	PUMP_STATUS:	(* Status and Fault *)
		Modbus.MB_Lock := TRUE;
		Modbus.MB_Query.SlaveAddress := Address;
		Modbus.MB_Query.FunctionCode := 3;
		ModBus.MB_Query.Read_StartAddress := 201;
		ModBus.MB_Query.Read_Quantity := 2;
		ModBus.MB_Start := TRUE;

		state := PUMP_DATA;

	PUMP_DATA:	(* Pump data *)
		IF NOT ModBus.MB_Start THEN
			IF ModBus.MB_MASTER.bInterfaceError<>0 OR ModBus.MB_MASTER.MB_Error<>0 THEN
				state := ERROR_STATE;
			ELSE
				DataPump.PumpStatus := ModBus.MB_Resp.Data[0];
				DataPump.PumpFault	:= WORD_TO_BOOL(ModBus.MB_Resp.Data[1]);

				ModBus.MB_Query.Read_StartAddress := 210;
				ModBus.MB_Query.Read_Quantity := 12;
				ModBus.MB_Start := TRUE;

				state := PUMP_ALARMS;
			END_IF
		END_IF

	PUMP_ALARMS: (* Historical alarms *)
		IF NOT ModBus.MB_Start THEN
			IF ModBus.MB_MASTER.bInterfaceError<>0 OR ModBus.MB_MASTER.MB_Error<>0 THEN
				state := ERROR_STATE;
			ELSE
				DataPump.PumpBoardTemp 	:= WORD_TO_INT(ModBus.MB_Resp.Data[0]);
				DataPump.PumpVoltage	:= ModBus.MB_Resp.Data[2];
				DataPump.PumpCurrent	:= ModBus.MB_Resp.Data[3];
				DataPump.PumpRPM		:= ModBus.MB_Resp.Data[5];
				DataPump.PumpPower		:= ModBus.MB_Resp.Data[6];
				DataPump.PumpOpTime		:= BUILD_16TO32(ADR(ModBus.MB_Resp.Data[7]));
				DataPump.PumpHead		:= ModBus.MB_Resp.Data[9];
				DataPump.PumpFlow		:= ModBus.MB_Resp.Data[10];
				DataPump.PumpLiqTemp	:= WORD_TO_INT(ModBus.MB_Resp.Data[11]);


				ModBus.MB_Query.Read_StartAddress := 230;
				ModBus.MB_Query.Read_Quantity := 15;
				ModBus.MB_Start := TRUE;

				state := PUMP_END_READ;
			END_IF
		END_IF

	PUMP_END_READ:	(* Read alarms *)
		IF NOT ModBus.MB_Start THEN
			IF ModBus.MB_MASTER.bInterfaceError<>0 OR ModBus.MB_MASTER.MB_Error<>0 THEN
				state := ERROR_STATE;
			ELSE
				DataPump.PumpAlarm[0] := ModBus.MB_Resp.Data[0];
				DataPump.PumpAlarm[1] := ModBus.MB_Resp.Data[1];
				DataPump.PumpAlarm[2] := ModBus.MB_Resp.Data[2];
				DataPump.PumpAlarm[3] := ModBus.MB_Resp.Data[3];
				DataPump.PumpAlarm[4] := ModBus.MB_Resp.Data[4];
				DataPump.PumpAlarm[5] := ModBus.MB_Resp.Data[5];
				DataPump.PumpAlarm[6] := ModBus.MB_Resp.Data[6];
				DataPump.PumpAlarm[7] := ModBus.MB_Resp.Data[7];
				DataPump.PumpAlarm[8] := ModBus.MB_Resp.Data[8];
				DataPump.PumpAlarm[9] := ModBus.MB_Resp.Data[9];
				DataPump.PumpAlarm[10] := ModBus.MB_Resp.Data[10];
				DataPump.PumpAlarm[11] := ModBus.MB_Resp.Data[11];
				DataPump.PumpAlarm[12] := ModBus.MB_Resp.Data[12];
				DataPump.PumpAlarm[13] := ModBus.MB_Resp.Data[13];
				DataPump.PumpAlarm[14] := ModBus.MB_Resp.Data[14];

				IF fModbusAlr THEN fModbusAlr := FALSE; END_IF

				ModBus.MB_Lock := FALSE;
				retry := 0;
				state := WAIT_STATE;

			END_IF
		END_IF

	(**** WRITE ON/OFF REGISTER AND VERIFY RIGHT SETTING ****)
	CIR_ON_OFF:	(* Pump On/off *)
		Modbus.MB_Lock := TRUE;
		Modbus.MB_Query.SlaveAddress := Address;
		Modbus.MB_Query.FunctionCode := 6;
		ModBus.MB_Query.Write_StartAddress := 110;
		ModBus.MB_Query.Write_Quantity := 1;
		ModBus.MB_Query.Write_Data[0] := BYTE_TO_WORD(Status);
		ModBus.MB_Start := TRUE;

		state := CIR_END_WRITE;

	CIR_END_WRITE:
		IF NOT ModBus.MB_Start THEN
			IF ModBus.MB_MASTER.bInterfaceError<>0 OR ModBus.MB_MASTER.MB_Error<>0 THEN
				state := ERROR_STATE;
			ELSE
				ModBus.MB_Lock := FALSE;
				retry := 0;
				state := WAIT_STATE;
				fWrite := FALSE;
			END_IF
		END_IF


	(**** CHECK MODBUS ERROR ****)
	ERROR_STATE: 	(* Release MODBUS *)
			MODBUS.MB_Lock:=FALSE;

			(* Retries *)
			retry:=retry+1;
			IF retry>3 THEN
				retry:=0;
				(* Signal event *)
				fModbusAlr := TRUE;
			END_IF

			state:=WAIT_STATE;
END_CASE
END_ACTION

(* POU Utils Functions/TONOF, ST *)
FUNCTION_BLOCK TONOF
VAR_INPUT
	IN		: BOOL;
	PT_ON	: TIME; (* time to pass, before OUT is set *)
	PT_OF	: TIME; (* time to pass, before OUT is reset *)
END_VAR
VAR_OUTPUT
	OUT		: BOOL;
END_VAR
VAR
	timer	: TON;
END_VAR
IF IN<>OUT THEN
	timer(IN:=TRUE,PT:=SEL(IN,PT_OF,PT_ON));
	IF timer.Q THEN OUT:=IN; END_IF
ELSE
	timer(IN:=FALSE);
END_IF
END_FUNCTION_BLOCK

(* POU Plant_Objects/obj_MODBUS_CIR_DOPPIO, ST *)
FUNCTION_BLOCK obj_MODBUS_CIR_DOPPIO
VAR CONSTANT
	WAIT_STATE		:	BYTE := 0;
	PUMP1_STATUS	:	BYTE := 1;
	PUMP1_DATA		:	BYTE := 2;
	PUMP1_ALARMS	:	BYTE := 3;
	PUMP1_END_READ	:	BYTE := 4;
	PUMP2_STATUS	:	BYTE := 5;
	PUMP2_DATA		:	BYTE := 6;
	PUMP2_ALARMS	:	BYTE := 7;
	PUMP2_END_READ	:	BYTE := 8;
	CIR_ON_OFF		:	BYTE := 90;
	CIR_ON_OFF_CHECK:	BYTE := 91;
	CIR_END_WRITE	:	BYTE := 92;
	ERROR_STATE		:	BYTE := 100;

	OFF				:	BYTE := 0;
	ON				:	BYTE := 1;
	ANTIFREEZE		:	BYTE := 2;
END_VAR
VAR_INPUT
	ID		:	BYTE;
	Address1:	BYTE;		(* Pump 1 address *)
	Address2:	BYTE;		(* Pump 2 address *)

	(* Physical inputs *)
	CIR_RUN_REQ		: BOOL; (* External run request (no heat or cold requested) *)
	CIR_STOP_REQ	: BOOL; (* External stop request (has priority over RUN signals!) *)
	PumpA_AL		: BOOL; (* Alarm input signal *)
	PumpB_AL		: BOOL;
	PumpA_AUTO		: BOOL;
	PumpB_AUTO		: BOOL;

	(* Controls *)
	OnOff			: BYTE;
END_VAR
VAR_IN_OUT
	ModBus		:	obj_MODBUS;
END_VAR
VAR_OUTPUT
	Run			:	BOOL;

	Status_Log	:	WORD;
	Status_Vis	:	DWORD;
END_VAR
VAR
	Ctrl_Run	:	BOOL;		(* Logical status of the device: 0: Not running (switched off), 1: running *)
	fWrite		:	BOOL;
	Status		:	BYTE;
	CIR_AUTO	:	BOOL;

	fStatus		:	FLT_EVENT;
	fCIR_AUTO	:	FLT_EVENT;

	DataPump1	:	typ_MODBUS_CIR;
	DataPump2	:	typ_MODBUS_CIR;
	Delay		: 	TONOF := (PT_OF:=Plant_CirOffDelay);

	state		:	BYTE;
	retry		:	BYTE;
	ReadTmr		:	TON := (PT:=T#5m);
	fModbusAlr	: 	BOOL;

	AlarmCtr	:	BYTE;
	WarningCtr	:	BYTE;

	AlarmHw1	:	FLT_EVENT := (INITEV:=FALSE);
	AlarmHw2	:	FLT_EVENT := (INITEV:=FALSE);
	Alarm1		:	FLT_EVENT := (INITEV:=FALSE);
	Alarm2		:	FLT_EVENT := (INITEV:=FALSE);
	Inverter1	:	FLT_EVENT := (INITEV:=FALSE);
	Inverter2	:	FLT_EVENT := (INITEV:=FALSE);
	ModbusAlr	:	FLT_EVENT := (INITEV:=FALSE);

	OldAlarmPump1	:	WORD;
	OldAlarmPump2	:	WORD;
	OldStatus	:	BYTE;

END_VAR
ManagePump();

(* State machine to read pump parameters *)
Stm();

(* Check alarm and warning for both pumps *)
CheckFault();

(* Set output according to logical On/Off status *)
IF AlarmCtr>0 THEN Run := FALSE;
ELSE Run := Ctrl_Run;
END_IF

IF AlarmCtr>0 THEN
	Status_Log := 2;
	Status_Vis := COLOR_RED;
ELSIF WarningCtr>0 THEN
	Status_Log := 1;
	Status_Vis := COLOR_YELLOW;
ELSE
	Status_Log := 0;
	Status_Vis := COLOR_GREEN;
END_IF

(* Update error lamp status *)
Lamp.UpdateStatus(obj_Status := Status_Log);
END_FUNCTION_BLOCK
ACTION AddLogData:
Logger.s1:=INSERT('&CIR=',BYTE_TO_STRING(ID),4);
IF ID<10 THEN Logger.s1:=INSERT(Logger.s1,'0',4); END_IF

(* PUMP 1 *)
Logger.s1:=CONCAT(Logger.s1,WORD_TO_STRING(DataPump1.PumpStatus));		Logger.s1:=CONCAT(Logger.s1,';');
Logger.s1:=CONCAT(Logger.s1,INT_TO_STRING(DataPump1.PumpBoardTemp));	Logger.s1:=CONCAT(Logger.s1,';');
Logger.s1:=CONCAT(Logger.s1,WORD_TO_STRING(DataPump1.PumpVoltage));		Logger.s1:=CONCAT(Logger.s1,';');
Logger.s1:=CONCAT(Logger.s1,WORD_TO_STRING(DataPump1.PumpRPM));			Logger.s1:=CONCAT(Logger.s1,';');
Logger.s1:=CONCAT(Logger.s1,WORD_TO_STRING(DataPump1.PumpPower));		Logger.s1:=CONCAT(Logger.s1,';');
Logger.s1:=CONCAT(Logger.s1,DWORD_TO_STRING(DataPump1.PumpOpTime));		Logger.s1:=CONCAT(Logger.s1,';');
Logger.s1:=CONCAT(Logger.s1,WORD_TO_STRING(DataPump1.PumpHead));		Logger.s1:=CONCAT(Logger.s1,';');
Logger.s1:=CONCAT(Logger.s1,WORD_TO_STRING(DataPump1.PumpFlow));		Logger.s1:=CONCAT(Logger.s1,';');
Logger.s1:=CONCAT(Logger.s1,WORD_TO_STRING(DataPump1.PumpLiqTemp));		Logger.s1:=CONCAT(Logger.s1,';');

(* PUMP 2 *)
Logger.s1:=CONCAT(Logger.s1,WORD_TO_STRING(DataPump2.PumpStatus));		Logger.s1:=CONCAT(Logger.s1,';');
Logger.s1:=CONCAT(Logger.s1,INT_TO_STRING(DataPump2.PumpBoardTemp));	Logger.s1:=CONCAT(Logger.s1,';');
Logger.s1:=CONCAT(Logger.s1,WORD_TO_STRING(DataPump2.PumpVoltage));		Logger.s1:=CONCAT(Logger.s1,';');
Logger.s1:=CONCAT(Logger.s1,WORD_TO_STRING(DataPump2.PumpRPM));			Logger.s1:=CONCAT(Logger.s1,';');
Logger.s1:=CONCAT(Logger.s1,WORD_TO_STRING(DataPump2.PumpPower));		Logger.s1:=CONCAT(Logger.s1,';');
Logger.s1:=CONCAT(Logger.s1,DWORD_TO_STRING(DataPump2.PumpOpTime));		Logger.s1:=CONCAT(Logger.s1,';');
Logger.s1:=CONCAT(Logger.s1,WORD_TO_STRING(DataPump2.PumpHead));		Logger.s1:=CONCAT(Logger.s1,';');
Logger.s1:=CONCAT(Logger.s1,WORD_TO_STRING(DataPump2.PumpFlow));		Logger.s1:=CONCAT(Logger.s1,';');
Logger.s1:=CONCAT(Logger.s1,WORD_TO_STRING(DataPump2.PumpLiqTemp));		Logger.s1:=CONCAT(Logger.s1,';');

Logger.s1:=CONCAT(Logger.s1,WORD_TO_STRING(Status_Log));
ADDSTRING(ADR(Logger.TData), ADR(Logger.s1), Logger.TLen);
END_ACTION
ACTION CheckFault:
(*** WARNINGS ***)

(* Verify ModBus error	*)
ModbusAlr(IN:=fModbusAlr);

IF ModbusAlr.EVH THEN
	LogEv(EL_Wrn,EO_CIRD,ID,23,SEL(ModBus.MB_MASTER.MB_Error<>0,'0','1'));
	WarningCtr := 1;
END_IF

IF ModbusAlr.EVL THEN WarningCtr := 0; END_IF


(*** ALARMS ***)

(**** PUMP 1 ****)

(* Hardware alarm (physical input *)
AlarmHw1(IN:=PumpA_AL);

IF AlarmHw1.EVH THEN
	LogEv(EL_Alarm,EO_CIRD,ID,3,'CIR_Alarm_A');
	AlarmCtr := AlarmCtr + 1;
END_IF

IF AlarmHw1.EVL THEN
	LogEv(EL_Log,EO_CIRD,ID,4,'CIR_Alarm_A_Recovered');
	AlarmCtr := AlarmCtr - 1;
END_IF

(* General alarm (read by Modbus) *)
Alarm1(IN:=(DataPump1.PumpAlarm[0] <> OldAlarmPump1));

IF Alarm1.EVH THEN
	IF DataPump1.PumpAlarm[0] = 0 THEN
		LogEv(EL_Alarm,EO_CIRD,ID,18,'Alarm_A_Recovered');
		AlarmCtr := AlarmCtr - 1;
	ELSE
		LogEv(EL_Alarm,EO_CIRD,ID,17,WORD_TO_STRING(DataPump1.PumpAlarm[0]));
		AlarmCtr := AlarmCtr + 1;
	END_IF

	OldAlarmPump1 := DataPump1.PumpAlarm[0];
END_IF

(* Inverter pump error *)
Inverter1(IN:=DataPump1.PumpFault);

IF Inverter1.EVH THEN
	LogEv(EL_Alarm,EO_CIRD,ID,15,'Inverter_Fault_A');
	AlarmCtr := AlarmCtr + 1;
END_IF

IF Inverter1.EVL THEN
	LogEv(EL_Alarm,EO_CIRD,ID,16,'Inverter_Fault_A_Recovered');
	AlarmCtr := AlarmCtr - 1;
END_IF


(**** PUMP 2 ****)

(* Hardware alarm (physical input *)
AlarmHw2(IN:=PumpB_AL);

IF AlarmHw2.EVH THEN
	LogEv(EL_Alarm,EO_CIRD,ID,11,'CIR_Alarm_B');
	AlarmCtr := AlarmCtr + 1;
END_IF

IF AlarmHw2.EVL THEN
	LogEv(EL_Log,EO_CIRD,ID,12,'CIR_Alarm_B_Recovered');
	AlarmCtr := AlarmCtr - 1;
END_IF

(* General alarm (read by Modbus) *)
Alarm2(IN:=(DataPump2.PumpAlarm[0] <> OldAlarmPump2));

IF Alarm2.EVH THEN
	IF DataPump2.PumpAlarm[0] = 0 THEN
		LogEv(EL_Log,EO_CIRD,ID,22,'Alarm_B_Recovered');
		AlarmCtr := AlarmCtr - 1;
	ELSE
		LogEv(EL_Alarm,EO_CIRD,ID,21,WORD_TO_STRING(DataPump2.PumpAlarm[0]));
		AlarmCtr := AlarmCtr + 1;
	END_IF

	OldAlarmPump2 := DataPump2.PumpAlarm[0];
END_IF

(* Inverter pump error *)
Inverter2(IN:=DataPump2.PumpFault);

IF Inverter2.EVH THEN
	LogEv(EL_Alarm,EO_CIRD,ID,19,'Inverter_Fault_B');
	AlarmCtr := AlarmCtr + 1;
END_IF

IF Inverter2.EVL THEN
	LogEv(EL_Log,EO_CIRD,ID,20,'Inverter_Fault_B_Recovered');
	AlarmCtr := AlarmCtr - 1;
END_IF
END_ACTION
ACTION ManagePump:
(*** Check if working in automatic (CIR_AUTO=1) or manual mode (CIR_AUTO=0) ***)
CIR_AUTO := PumpA_AUTO OR PumpB_AUTO;

fCIR_AUTO(IN:=CIR_AUTO);

(* MANUAL MODE *)
IF fCIR_AUTO.EVL THEN
	LogEv(EL_Wrn,EO_CIR,ID,7,'CIR_Manual');
	Status := 2;
END_IF

IF fCIR_AUTO.EVH THEN LogEv(EL_Log,EO_CIRD,ID,8,'CIR_Auto'  ); END_IF

(* AUTOMATIC MODE *)
IF CIR_AUTO THEN

	CASE OnOff OF

		OFF:
			(* Switch off pump *)
			Ctrl_Run := FALSE;			(* Logically swtched off *)
			Delay(IN:=Ctrl_Run);		(* Count delay time before physical switch off	*)

		ON:
			(* Switch on pump *)
			Delay(IN:=TRUE, PT_ON:=WORD_TO_TIME(1000*ID));	(* Start switch on delay time - proportional to object id *)

			(* Set logical running variable as true -> CIR running *)
			IF (NOT Ctrl_Run AND Delay.OUT) THEN Ctrl_Run := TRUE;	END_IF

		ANTIFREEZE:
			(* Antifreeze condition: switch on pump without change logical status ("Ctrl_Run" kept false)	*)
			Delay(IN:=TRUE, PT_ON:=T#0s);		(* Antifreeze -> Enable immediatly *)

	END_CASE

	(* Verify if a forced condition is request *)
	IF CIR_STOP_REQ    THEN Status := 0;
	ELSIF CIR_RUN_REQ  THEN Status := 1;
	ELSE Status := BOOL_TO_BYTE(Delay.OUT);
	END_IF

	(* If functioning status has changed, phisically modify it according to variable state, otherwise keep same status *)
	fStatus(IN:=(Status<>OldStatus));

	IF fStatus.EVH THEN
		fWrite := TRUE;
		OldStatus := Status;
	END_IF

END_IF
END_ACTION
ACTION Stm:
CASE state OF
	WAIT_STATE:	(* Refresh time manager *)
		ReadTmr(IN:=NOT ReadTmr.Q);
		IF ReadTmr.Q THEN
			state := PUMP1_STATUS;
			ReadTmr.PT := T#1m;
		END_IF

		IF fWrite THEN state := CIR_ON_OFF;	END_IF

	(**** READ CIR PARAMETERS ****)

	(**** PUMP 1 ****)
	PUMP1_STATUS:	(* Status and Fault *)
		Modbus.MB_Lock := TRUE;
		Modbus.MB_Query.SlaveAddress := Address1;
		Modbus.MB_Query.FunctionCode := 3;
		ModBus.MB_Query.Read_StartAddress := 201;
		ModBus.MB_Query.Read_Quantity := 2;
		ModBus.MB_Start := TRUE;

		state := PUMP1_DATA;

	PUMP1_DATA:	(* Pump data *)
		IF NOT ModBus.MB_Start THEN
			IF ModBus.MB_MASTER.bInterfaceError<>0 THEN
				state := ERROR_STATE;
			ELSE
				DataPump1.PumpStatus := ModBus.MB_Resp.Data[0];
				DataPump1.PumpFault	:= WORD_TO_BOOL(ModBus.MB_Resp.Data[1]);

				ModBus.MB_Query.Read_StartAddress := 210;
				ModBus.MB_Query.Read_Quantity := 12;
				ModBus.MB_Start := TRUE;

				state := PUMP1_ALARMS;
			END_IF
		END_IF

	PUMP1_ALARMS: (* Historical alarms *)
		IF NOT ModBus.MB_Start THEN
			IF ModBus.MB_MASTER.bInterfaceError<>0 THEN
				state := ERROR_STATE;
			ELSE
				DataPump1.PumpBoardTemp := WORD_TO_INT(ModBus.MB_Resp.Data[0]);
				DataPump1.PumpVoltage	:= ModBus.MB_Resp.Data[2];
				DataPump1.PumpCurrent	:= ModBus.MB_Resp.Data[3];
				DataPump1.PumpRPM		:= ModBus.MB_Resp.Data[5];
				DataPump1.PumpPower		:= ModBus.MB_Resp.Data[6];
				DataPump1.PumpOpTime	:= BUILD_16TO32(ADR(ModBus.MB_Resp.Data[7]));
				DataPump1.PumpHead		:= ModBus.MB_Resp.Data[9];
				DataPump1.PumpFlow		:= ModBus.MB_Resp.Data[10];
				DataPump1.PumpLiqTemp	:= WORD_TO_INT(ModBus.MB_Resp.Data[11]);


				ModBus.MB_Query.Read_StartAddress := 230;
				ModBus.MB_Query.Read_Quantity := 15;
				ModBus.MB_Start := TRUE;

				state := PUMP1_END_READ;
			END_IF
		END_IF

	PUMP1_END_READ:	(* Read alarms *)
		IF NOT ModBus.MB_Start THEN
			IF ModBus.MB_MASTER.bInterfaceError<>0 THEN
				state := ERROR_STATE;
			ELSE
				DataPump1.PumpAlarm[0] := ModBus.MB_Resp.Data[0];
				DataPump1.PumpAlarm[1] := ModBus.MB_Resp.Data[1];
				DataPump1.PumpAlarm[2] := ModBus.MB_Resp.Data[2];
				DataPump1.PumpAlarm[3] := ModBus.MB_Resp.Data[3];
				DataPump1.PumpAlarm[4] := ModBus.MB_Resp.Data[4];
				DataPump1.PumpAlarm[5] := ModBus.MB_Resp.Data[5];
				DataPump1.PumpAlarm[6] := ModBus.MB_Resp.Data[6];
				DataPump1.PumpAlarm[7] := ModBus.MB_Resp.Data[7];
				DataPump1.PumpAlarm[8] := ModBus.MB_Resp.Data[8];
				DataPump1.PumpAlarm[9] := ModBus.MB_Resp.Data[9];
				DataPump1.PumpAlarm[10] := ModBus.MB_Resp.Data[10];
				DataPump1.PumpAlarm[11] := ModBus.MB_Resp.Data[11];
				DataPump1.PumpAlarm[12] := ModBus.MB_Resp.Data[12];
				DataPump1.PumpAlarm[13] := ModBus.MB_Resp.Data[13];
				DataPump1.PumpAlarm[14] := ModBus.MB_Resp.Data[14];

				state := PUMP2_STATUS;
			END_IF
		END_IF

	(**** PUMP 2 ****)
	PUMP2_STATUS:	(* Status and Fault *)
		Modbus.MB_Lock := TRUE;
		Modbus.MB_Query.SlaveAddress := Address2;
		Modbus.MB_Query.FunctionCode := 3;
		ModBus.MB_Query.Read_StartAddress := 201;
		ModBus.MB_Query.Read_Quantity := 2;
		ModBus.MB_Start := TRUE;

		state := PUMP2_DATA;

	PUMP2_DATA:	(* Pump data *)
		IF NOT ModBus.MB_Start THEN
			IF ModBus.MB_MASTER.bInterfaceError<>0 THEN
				state := ERROR_STATE;
			ELSE
				DataPump2.PumpStatus := ModBus.MB_Resp.Data[0];
				DataPump2.PumpFault	:= WORD_TO_BOOL(ModBus.MB_Resp.Data[1]);

				ModBus.MB_Query.Read_StartAddress := 210;
				ModBus.MB_Query.Read_Quantity := 12;
				ModBus.MB_Start := TRUE;

				state := PUMP2_ALARMS;
			END_IF
		END_IF

	PUMP2_ALARMS:
		IF NOT ModBus.MB_Start THEN
			IF ModBus.MB_MASTER.bInterfaceError<>0 THEN
				state := ERROR_STATE;
			ELSE
				DataPump2.PumpBoardTemp := WORD_TO_INT(ModBus.MB_Resp.Data[0]);
				DataPump2.PumpVoltage	:= ModBus.MB_Resp.Data[2];
				DataPump2.PumpCurrent	:= ModBus.MB_Resp.Data[3];
				DataPump2.PumpRPM		:= ModBus.MB_Resp.Data[5];
				DataPump2.PumpPower		:= ModBus.MB_Resp.Data[6];
				DataPump2.PumpOpTime	:= BUILD_16TO32(ADR(ModBus.MB_Resp.Data[7]));
				DataPump2.PumpHead		:= ModBus.MB_Resp.Data[9];
				DataPump2.PumpFlow		:= ModBus.MB_Resp.Data[10];
				DataPump2.PumpLiqTemp	:= WORD_TO_INT(ModBus.MB_Resp.Data[11]);


				ModBus.MB_Query.Read_StartAddress := 230;
				ModBus.MB_Query.Read_Quantity := 15;
				ModBus.MB_Start := TRUE;

				state := PUMP2_END_READ;
			END_IF
		END_IF

	PUMP2_END_READ:
		IF NOT ModBus.MB_Start THEN
			IF ModBus.MB_MASTER.bInterfaceError<>0 THEN
				state := ERROR_STATE;
			ELSE
				DataPump2.PumpAlarm[0] := ModBus.MB_Resp.Data[0];
				DataPump2.PumpAlarm[1] := ModBus.MB_Resp.Data[1];
				DataPump2.PumpAlarm[2] := ModBus.MB_Resp.Data[2];
				DataPump2.PumpAlarm[3] := ModBus.MB_Resp.Data[3];
				DataPump2.PumpAlarm[4] := ModBus.MB_Resp.Data[4];
				DataPump2.PumpAlarm[5] := ModBus.MB_Resp.Data[5];
				DataPump2.PumpAlarm[6] := ModBus.MB_Resp.Data[6];
				DataPump2.PumpAlarm[7] := ModBus.MB_Resp.Data[7];
				DataPump2.PumpAlarm[8] := ModBus.MB_Resp.Data[8];
				DataPump2.PumpAlarm[9] := ModBus.MB_Resp.Data[9];
				DataPump2.PumpAlarm[10] := ModBus.MB_Resp.Data[10];
				DataPump2.PumpAlarm[11] := ModBus.MB_Resp.Data[11];
				DataPump2.PumpAlarm[12] := ModBus.MB_Resp.Data[12];
				DataPump2.PumpAlarm[13] := ModBus.MB_Resp.Data[13];
				DataPump2.PumpAlarm[14] := ModBus.MB_Resp.Data[14];

				IF fModbusAlr THEN fModbusAlr := FALSE; END_IF

				ModBus.MB_Lock := FALSE;
				retry := 0;
				state := WAIT_STATE;

			END_IF
		END_IF

	(**** WRITE ON/OFF REGISTER AND VERIFY RIGHT SETTING ****)
	CIR_ON_OFF:	(* Pump On/off *)
		Modbus.MB_Lock := TRUE;
		Modbus.MB_Query.SlaveAddress := Address1;
		Modbus.MB_Query.FunctionCode := 6;
		ModBus.MB_Query.Write_StartAddress := 110;
		ModBus.MB_Query.Write_Quantity := 1;
		ModBus.MB_Query.Write_Data[0] := BYTE_TO_WORD(Status);
		ModBus.MB_Start := TRUE;

		state := CIR_END_WRITE;

	CIR_END_WRITE:
		IF NOT ModBus.MB_Start THEN
			IF ModBus.MB_MASTER.bInterfaceError<>0 THEN
				state := ERROR_STATE;
			ELSE
				ModBus.MB_Lock := FALSE;
				retry := 0;
				state := WAIT_STATE;
				fWrite := FALSE;
			END_IF
		END_IF


	(**** CHECK MODBUS ERROR ****)
	ERROR_STATE: 	(* Release MODBUS *)
			MODBUS.MB_Lock:=FALSE;

			(* Retries *)
			retry:=retry+1;
			IF retry>3 THEN
				retry:=0;
				(* Signal event *)
				fModbusAlr := TRUE;
			END_IF

			state:=WAIT_STATE;
END_CASE
END_ACTION

(* POU Plant_Objects/obj_MODBUS_TCP, ST *)
FUNCTION_BLOCK obj_MODBUS_TCP
(* === MODBUS-TCP PROTOCOL INTERFACE ===
   v1.0[10/06/15] - Create
*)
VAR CONSTANT
	VARS_Max	: BYTE := 32;
END_VAR
VAR_INPUT
	(* Settings *)
	ID			: BYTE;
	IP			: STRING;
	PORT		: WORD:=502;
	(* Interface *)
	MB_MASTER	: ETHERNET_MODBUSMASTER_TCP;
	MB_READBUF	: ARRAY [0..128] OF WORD;
	MB_WRITEBUF : ARRAY [0..128] OF WORD;
	MB_Start	: BOOL;
	MB_Lock		: BOOL;
	(* Variables management *)
	VARS_En		: BOOL;
	VARS		: ARRAY [0..VARS_Max] OF typ_MODBUS_VAR;
	VARS_Check	: BOOL;
	VARS_Alarm	: BOOL;
	(* Variables allocation *)
	VAR_Pointer : POINTER TO ARRAY[0..99] OF WORD;
	VAR_Cfg		: POINTER TO typ_MODBUS_VAR;
END_VAR
VAR_OUTPUT
	(* Status *)
	Status_Log	: BYTE;
	Status_Vis	: DWORD;
END_VAR
VAR
	sta         : BYTE :=0;
	i			: BYTE;
	j			: BYTE;
	Alarm		: FLT_EVENT;

	VarTmr		: TON := (PT:=T#1s);
	VarSta		: BYTE; (* Status *)
	VarCnt		: BYTE; (* Scan counter *)
	VarRetry	: BYTE;
	VarAlarm	: BYTE; (* Last variable with errors *)
END_VAR
MB_MASTER( strIP_ADDRESS:=IP, wPORT:=PORT, tTIME_OUT:=T#750MS, (*xCONNECT:=TRUE,*)
		   ptREAD_DATA:=ADR(MB_READBUF), ptSEND_DATA:=ADR(MB_WRITEBUF), xSEND:=MB_Start );

IF sta=0 THEN
	MB_MASTER.xCONNECT:=TRUE;
	sta:=1;
END_IF

(* Process variable management *)
IF VARS_En THEN VARS_Process(); END_IF

(* Check status *)
Alarm(IN:=(MB_MASTER.wERROR<>0));
IF Alarm.EVH THEN
	LogEv(SEL(MB_MASTER.wERROR>0,EL_Wrn,EL_Alarm),EO_MODBUS_TCP,ID,1,WORD_TO_STRING(MB_MASTER.wERROR));
END_IF
IF Alarm.EVL THEN
	LogEv(EL_Log,EO_MODBUS_TCP,ID,2,'');
END_IF

(* Log/visu status *)
   IF Alarm.IN   THEN Status_Log:=2; Status_Vis:=COLOR_RED;
ELSIF Vars_Alarm THEN Status_Log:=1; Status_Vis:=COLOR_YELLOW;
  				 ELSE Status_Log:=0; Status_Vis:=COLOR_GREEN;
END_IF
END_FUNCTION_BLOCK
ACTION VAR_Search:
(* Search VAR with specific pointer if not found return first free VAR
	[Last VAR is not active... used as safe area...] 
*)
j:=VARS_Max;
FOR i := 0 TO VARS_Max-1 DO
	IF VARS[i].Variable=0 AND j>i THEN j:=i; END_IF
	IF VARS[i].Variable=VAR_Pointer THEN
		VAR_Cfg:=ADR(VARS[i]);
		RETURN;
	END_IF
END_FOR
VAR_Cfg:=ADR(VARS[j]);
END_ACTION
ACTION VARS_Process:
(* Update var timers *)
VarTmr(IN:=(NOT VarTmr.Q));
IF VarTmr.Q THEN
	FOR i := 0 TO VARS_Max DO
		IF VARS[i].Refresh_Cnt>0 THEN VARS[i].Refresh_Cnt:=VARS[i].Refresh_Cnt-1; END_IF
	END_FOR
	VARS_Check:=TRUE;
END_IF


(* Process status *)
CASE VarSta OF
	0: (* === Init *)
		VarCnt:=0;
		VarSta:=1;

	1: (* === Wait check signal *)
		IF VARS_Check THEN
			VARS_Check:=FALSE;
			VarCnt:=0;
			VarSta:=2;
		END_IF

	2: (* === Check loop *)
		IF NOT (MB_Lock OR MB_Start) THEN
			WHILE VarCnt<=(VARS_Max-1) AND VarSta=2 DO
				(* Check only active vars *)
				IF VARS[VarCnt].Variable<>0 THEN
					(* Check var auto-refresh on timer checks *)
					IF VARS[VarCnt].Refresh_Time>0 AND VARS[VarCnt].Refresh_Cnt=0 THEN
						VARS[VarCnt].Refresh_Cnt:=VARS[VarCnt].Refresh_Time;
						VarSta:=3;
					END_IF
					(* Check refresh for change or request *)
					CASE VARS[VarCnt].FunCode OF
						5,6,15,16: (* Write functions *)
							IF VARS[VarCnt].Variable_Size=1 THEN
								IF VARS[VarCnt].Variable^<>VARS[VarCnt].Variable_Mirror THEN
									VARS[VarCnt].Variable_Mirror:=VARS[VarCnt].Variable^;
									VarSta:=3;
								END_IF
							ELSE
								IF VARS[VarCnt].Variable_Mirror<>0 THEN
									VARS[VarCnt].Variable_Mirror:=0;
									VarSta:=3;
								END_IF
							END_IF
						1,2,3,4: (* Write functions *)
							IF VARS[VarCnt].Variable_Mirror<>0 THEN
								VARS[VarCnt].Variable_Mirror:=0;
								VarSta:=3;
							END_IF
					END_CASE
				END_IF
				(* Process query *)
				IF VarSta=3 THEN
					MB_Lock:=TRUE;
					MB_MASTER.bUNIT_ID:=VARS[VarCnt].SlaveAddress;
					MB_MASTER.bFUNCTION_CODE:=VARS[VarCnt].FunCode;
					CASE VARS[VarCnt].FunCode OF
						16#5,16#6,16#F,16#10:
							MB_MASTER.wREAD_ADDRESS:=0;
							MB_MASTER.wREAD_QUANTITY:=0;
							MB_MASTER.wWRITE_ADDRESS:=VARS[VarCnt].FunAddress;
							MB_MASTER.wWRITE_QUANTITY:=VARS[VarCnt].Variable_Size;
							IF VARS[VarCnt].Variable_Size=200 THEN
								COPY_32SWAP16(VARS[VarCnt].Variable, ADR(MB_WRITEBUF));
							ELSIF VARS[VarCnt].Variable_Size>1 THEN
								MEMCPY(VARS[VarCnt].Variable, ADR(MB_WRITEBUF), 2*VARS[VarCnt].Variable_Size);
							ELSE
								MB_WRITEBUF[0]:=VARS[VarCnt].Variable^;
							END_IF
						16#1,16#2,16#3,16#4:
							MB_MASTER.wREAD_ADDRESS:=VARS[VarCnt].FunAddress;
							IF VARS[VarCnt].Variable_Size=200 THEN MB_MASTER.wREAD_QUANTITY:=2; ELSE
							  MB_MASTER.wREAD_QUANTITY:=VARS[VarCnt].Variable_Size;
							END_IF
							MB_MASTER.wWRITE_ADDRESS:=0;
							MB_MASTER.wWRITE_QUANTITY:=0;
					END_CASE
					VarRetry:=0;
					MB_Start:=TRUE;
				ELSE
					VarCnt:=VarCnt+1;
				END_IF
			END_WHILE
			(* Check loop completed -> no actions *)
			IF VarSta=2 THEN VarSta:=1; END_IF
		END_IF

	3: (* === Wait & process MB response *)
		IF NOT MB_Start THEN
			IF MB_MASTER.wERROR=0 THEN
				CASE VARS[VarCnt].FunCode OF
					1,2,3,4:
						IF VARS[VarCnt].Variable_Size=200 THEN
							COPY_32SWAP16(ADR(MB_READBUF), VARS[VarCnt].Variable);
						ELSIF VARS[VarCnt].Variable_Size>1 THEN
							MEMCPY(ADR(MB_READBUF), VARS[VarCnt].Variable, 2*VARS[VarCnt].Variable_Size);
						ELSE
							VARS[VarCnt].Variable^:=MB_READBUF[0];
						END_IF
				END_CASE
				MB_Lock:=FALSE;
				(* Signal error recovery *)
				IF VARS_Alarm=TRUE AND VarCnt=VarAlarm THEN
					LogEv(EL_Wrn,EO_MODBUS_TCP,ID,5,'');
					VARS_Alarm:=FALSE;
				END_IF
				(* Next var *)
				VarCnt:=VarCnt+1;
				VarSta:=2;
			ELSE
				IF VarRetry<10 THEN
					VarRetry:=VarRetry+1;
					MB_Start:=TRUE;
				ELSE
					MB_Lock:=FALSE;
					(* Signal error *)
					IF VARS_Alarm=FALSE THEN
						LogEv(EL_Wrn,EO_MODBUS_TCP,ID,3,WORD_TO_STRING(MB_MASTER.wERROR));
						VARS_Alarm:=TRUE;
						VarAlarm:=VarCnt-1;
					END_IF
					(* Next var *)
					VarCnt:=VarCnt+1;
					VarSta:=2;
				END_IF
			END_IF
		END_IF

ELSE
	VarSta:=0;
END_CASE
END_ACTION

(* POU Plant_Objects/obj_TPV, ST *)
FUNCTION_BLOCK obj_TPV
(* === TEMPERATURE PROBE  ===
   v1.0[16/04/15] - Versioning
*)
VAR CONSTANT
	NormalEv		: BYTE := 0;
	ErrorEv			: BYTE := 1;
	WarningEv		: BYTE := 2;
END_VAR
VAR_INPUT
	(* Settings *)
	ID				: BYTE;
	TAP				: BYTE:=4;	   (* Consecutive checks filter *)
	INITEV			: BOOL:= TRUE; (* Generate init OK event *)
	IN_EMIN			: INT :=-2000; (* Low error limit *)
	IN_WMIN			: INT := -550; (* Low warning value *)
	IN_WMAX			: INT :=  900; (* High warning value *)
	IN_EMAX			: INT := 8500; (* High error limit *)
	ERR_MIN_SHORT	: BOOL:= TRUE; (* TRUE  ==> EMIN=Short        , EMAX=Disconnected
									  FALSE ==> EMIN=Disconnected , EMAX=Short 		 *)
	(* Physical input *)
	IN			: INT;
END_VAR
VAR_OUTPUT
	WRN			: BOOL;	(* Value in warning range *)
	ERR			: BOOL;	(* Value error *)
	HI			: INT;	(* Highest value - cleared by Stat_Reset() action *)
	AVG			: INT; 	(* Average value - updated by Mean() action, cleared by Mean_Reset() action *)
	LOW			: INT;	(* Lowest value  - cleared by Stat_Reset() action *)

	Status_Log	: WORD;
	Status_Vis	: DWORD;
END_VAR
VAR
	cnt			: BYTE;
	event		: BYTE := 0;	(* 0: monitoring a generic, 1: monitoring an error, 2: monitoring a warning *)
	asum		: DINT;
	acnt		: WORD;
END_VAR
(* Check probe value limits *)
IF IN<=IN_EMIN OR IN>=IN_EMAX THEN
	IF NOT ERR THEN
		IF event <> ErrorEv THEN
			cnt := 1;
			event := ErrorEv;
		ELSE
			cnt:=cnt+1;
		END_IF

		IF cnt>TAP THEN
			cnt:=0;
			ERR:=TRUE; WRN:=FALSE;
			IF ( ERR_MIN_SHORT=TRUE  AND IN<=IN_EMIN ) OR ( ERR_MIN_SHORT=FALSE AND IN>=IN_EMAX ) THEN
				LogEv(EL_Alarm,EO_TPV,ID,5,INT_TO_STRING(IN));
			ELSE
				LogEv(EL_Alarm,EO_TPV,ID,4,INT_TO_STRING(IN));
			END_IF
		END_IF
	END_IF
ELSIF IN<=IN_WMIN OR IN>=IN_WMAX THEN
	IF NOT WRN THEN
		IF event <> WarningEv THEN
			cnt := 1;
			event := WarningEv;
		ELSE
			cnt:=cnt+1;
		END_IF

		IF cnt>TAP THEN
			cnt:=0;
			ERR:=FALSE; WRN:=TRUE;
			LogEv(EL_Wrn,EO_TPV,ID,SEL(IN<=IN_WMIN,3,2),INT_TO_STRING(IN));
		END_IF
	END_IF
ELSE
	IF INITEV OR WRN OR ERR THEN
		IF event <> NormalEv THEN
			cnt := 1;
			event := NormalEv;
		ELSE
			cnt:=cnt+1;
		END_IF

		IF cnt>TAP THEN
			cnt:=0;
			INITEV:=FALSE; ERR:=FALSE; WRN:=FALSE;
			LogEv(EL_Log,EO_TPV,ID,1,'Probe_OK');
		END_IF
	END_IF
END_IF

(* Average value *)
IF acnt>=60000 THEN
	Mean();
	asum := asum - AVG;
	acnt := acnt - 1;
END_IF

asum := asum + IN;
acnt := acnt + 1;

(* Statistics values *)
IF IN<LOW THEN LOW:=IN; END_IF
IF IN>HI  THEN HI :=IN; END_IF

Lamp.obj_Status := Status_Log;
Lamp.UpdateStatus();

(* Status Log *)
IF ERR THEN	Status_Log := 2; Status_Vis := COLOR_RED;
ELSIF WRN THEN Status_Log := 1;	Status_Vis := COLOR_YELLOW;
ELSE Status_Log := 0; Status_Vis := COLOR_GREEN;
END_IF
END_FUNCTION_BLOCK
ACTION AddLogData:
Logger.s1:=INSERT('&TPV=',BYTE_TO_STRING(ID),4);
IF ID<10 THEN Logger.s1:=INSERT(Logger.s1,'0',4); END_IF

Mean();

Logger.s1:=CONCAT(Logger.s1,INT_TO_STRING(AVG));		Logger.s1:=CONCAT(Logger.s1,';');

Logger.s1:=CONCAT(Logger.s1,WORD_TO_STRING(Status_Log));
ADDSTRING(ADR(Logger.TData), ADR(Logger.s1), Logger.TLen);
END_ACTION
ACTION Mean:
AVG := DINT_TO_INT(asum/acnt);
END_ACTION
ACTION Mean_Reset:
AVG:=IN;
asum:=IN;
acnt:=1;
END_ACTION
ACTION Stat_Reset:
HI:=IN;
LOW:=IN;
END_ACTION

(* POU Plant_Objects/obj_VRD_ONOFF, ST *)
FUNCTION_BLOCK obj_VRD_ONOFF
(* === SERVOMOTORE APERTO/CHIUSO (ON/OFF) ===
   v1.0[04/08/15] - Create
*)
VAR CONSTANT
	INIT_COUNT	:	BYTE := 0;
	COUNTING	:	BYTE := 1;
	NORMAL		:	BYTE := 2;
END_VAR
VAR_INPUT
	ID			:	BYTE;

	SetPoint	:	INT;
	Feedback	:	BOOL;

	StrokeTime	:	TIME;	(* Time needed to drive through the entire stroke IN SECONDS!! *)
END_VAR
VAR_OUTPUT
	OUT_CL	:	BOOL;	(* Manage close phisical output *)
	OUT_OP	:	BOOL;	(* Manage open phisical output *)

	Status_Log	:	WORD;
	Status_Vis	:	DWORD;
END_VAR
VAR
	Status	:	BOOL;	(* TRUE: Valve open, FALSE: Valve close *)
	InitOK	:	BOOL;
	Delay	:	WORD;
	count	:	WORD;

	state	:	BYTE;

	Change	:	FLT_EVENT;
END_VAR
IF NOT InitOK THEN
	(* This object is called every 500ms, so total counter needs to be two times the value passed as input (expressed in seconds) *)
	Delay := TIME_TO_WORD(StrokeTime) * 2;
	InitOK := TRUE;
END_IF

(* Update valve position according to value passed as input *)
IF SetPoint > 1000 THEN

	(* Open valve *)
	OUT_CL := FALSE;
	OUT_OP := TRUE;

	Status := TRUE;

ELSE

	(* Open valve *)
	OUT_OP := FALSE;
	OUT_CL := TRUE;

	Status := FALSE;

END_IF

(* Check if a status change happens *)
Change(IN:=Status);

IF Change.EVH THEN state := INIT_COUNT; END_IF

(* State machine *)
Stm();

(* Status Log *)
IF Status_Log = 2 THEN Status_Vis := COLOR_RED;
ELSIF Status_Log = 1 THEN Status_Vis := COLOR_YELLOW;
ELSE Status_Vis := COLOR_GREEN;
END_IF

Lamp.UpdateStatus(obj_Status := Status_Log);
END_FUNCTION_BLOCK
ACTION Stm:
CASE state OF

	INIT_COUNT:	(* Init counting *)
		count := 0;
		state := COUNTING;

	COUNTING:	(* Wait state (1s tolerance on the counting) *)
		IF count < (Delay + 2) THEN
			count := count + 1;
		ELSE
			IF Feedback <> Status THEN
				LogEv(EL_Alarm,0,ID,2,'');
				Status_Log := 2;
			ELSE
				IF Status_Log = 2 THEN
					LogEv(EL_Log,0,ID,1,'');
					Status_Log := 0;
				END_IF
			END_IF

			state := NORMAL;
		END_IF

	NORMAL:(* Normal operation -> Do nothing *)
		(*state := NORMAL;*);

END_CASE
END_ACTION

(* POU Plant_Objects/obj_VRD_ONOFF_new, ST *)
FUNCTION_BLOCK obj_VRD_ONOFF_new
(* === SERVOMOTORE APERTO/CHIUSO (ON/OFF) ===
   v1.0[04/08/15] - Create
*)
VAR CONSTANT
	INIT_COUNT	:	BYTE := 0;
	COUNTING	:	BYTE := 1;
	NORMAL		:	BYTE := 2;
END_VAR
VAR_INPUT
	ID			:	BYTE;

	SetPoint	:	INT;
	Feedback	:	BOOL;

	StrokeTime	:	TIME;	(* Time needed to drive through the entire stroke IN SECONDS!! *)
END_VAR
VAR_OUTPUT
	(* Physical outputs *)
	OUT_CL	:	BOOL;	(* Manage close phisical output *)
	OUT_OP	:	BOOL;	(* Manage open phisical output *)

	Status_Log	:	WORD;
	Status_Vis	:	DWORD;
END_VAR
VAR
	Status		:	BOOL;	(* TRUE: Valve open, FALSE: Valve close *)
	fWait		:	BOOL;

	Timer		:	TON;

	Change		:	FLT_EVENT := (INITEV:=FALSE);
	chkStatus	:	FLT_EVENT := (INITEV:=FALSE);
END_VAR
(* Update valve position according to value passed as input *)
IF SetPoint > 1000 THEN
	(* Open valve *)
	OUT_CL := FALSE;
	OUT_OP := TRUE;

	Status := TRUE;
ELSE
	(* Close valve *)
	OUT_OP := FALSE;
	OUT_CL := TRUE;

	Status := FALSE;
END_IF

(* Check if a status change happens *)
Change(IN:=Status);

IF Change.EVH OR Change.EVL THEN fWait := TRUE; END_IF

IF fWait THEN
	Timer(IN:=Timer.Q, PT:=StrokeTime);
	
	IF Timer.Q THEN
		(* Check feedback *)
		chkStatus(IN:=(Status<>Feedback));
	
		IF chkStatus.EVH THEN
			LogEv(EL_Alarm,EO_VRD,ID,4,'');
			Status_Log := 0;
		END_IF
	
		IF chkStatus.EVL THEN Status_Log := 0; END_IF

		fWait := FALSE;
	END_IF
END_IF

(* Status Log *)
IF Status_Log = 2 THEN Status_Vis := COLOR_RED;
ELSIF Status_Log = 1 THEN Status_Vis := COLOR_YELLOW;
ELSE Status_Vis := COLOR_GREEN;
END_IF

Lamp.UpdateStatus(obj_Status := Status_Log);
END_FUNCTION_BLOCK

(* POU Plant_Objects/obj_ZTHL, ST *)
FUNCTION_BLOCK obj_ZTHL
(* === ZIGBEE AMBIENT SENSORS MT-200 ===
   v1.0[07/05/05] - Create
*)
VAR CONSTANT
	(* States *)
	WAIT_STATE			:	BYTE := 0;
	STATUS_REQUEST		:	BYTE := 1;
	LQI_REQUEST			:	BYTE := 2;
	MEAS_REQUEST		:	BYTE := 3;
	END_READ			:	BYTE := 4;
	ERROR_STATE			:	BYTE := 100;

	LQI_Threshold		:	WORD := 100;		(* Zigbee link quality minimum value *)
	LowBattVoltage		:	WORD := 270;		(* Battery is considered low when reaches 1.35V each *)
END_VAR
VAR_INPUT
	(* Settings *)
	ID				: BYTE;
	Address			: BYTE;

	Refresh_Period	: TIME:=t#5m;
	(* Controls *)
	Refresh_Auto	: BOOL:=TRUE; (* Enable automatic refresh *)
	Refresh_Now		: BOOL; 	  (* Force an immediate refresh *)

	(* Limits *)
	Tmin			: INT := 0;
	Tmax			: INT := 400;
END_VAR
VAR_IN_OUT
	(* Interface *)
	MODBUS			: obj_MODBUS_TCP;
END_VAR
VAR_OUTPUT
	OUT_TEMP		: INT;	(* Temperatura misurata [°C/10] *)
	OUT_HYGRO		: INT;	(* Umidità misurata [%] *)
	OUT_LUX			: INT;	(* Luce misurata [lux] *)
	OUT_VBATT		: INT;	(* Tensione misurata dalla batteria [V/100] *)

	OUT_LQI			: BYTE;

	ERR				: BOOL;

	fTemp			: BOOL;

	(* Status *)
	Status_Log		: BYTE;
	Status_Vis 		: DWORD;
END_VAR
VAR
	dly 	 		: TON := (PT:=t#5s);

	sta				: BYTE;
	retry	 		: BYTE;

	OldNodeStatus	: WORD;
	fLQI			: BOOL;
	fBatt			: BOOL;
	Quality			: FLT_EVENT := (INITEV:=FALSE);
	Battery			: FLT_EVENT;
	Temperature		: FLT_EVENT;
	Alarm			: FLT_EVENT;

	StatusOK		: BYTE;			(* 0: Status OK, >=1: Alarm and/or warning		Incremented by 1 when Alarm or Wrn occurs,
																					decremented by 1 when restored	*)
END_VAR
CASE sta OF
	WAIT_STATE: (* === Wait update signals *)
		dly(IN:=NOT (dly.Q OR Refresh_Now OR (NOT Refresh_Auto)));
		IF dly.Q OR Refresh_Now THEN
			dly.PT:=Refresh_Period;
			Refresh_Now:=FALSE;
			(*sta:=STATUS_REQUEST;*)
			sta:=LQI_REQUEST;
		END_IF

	STATUS_REQUEST:	(* Node status *)
		IF NOT (MODBUS.MB_Lock OR MODBUS.MB_Start) THEN
			MODBUS.MB_Lock:=TRUE;
			MODBUS.ID:=ID;
			MODBUS.MB_MASTER.bUNIT_ID := Address;
			MODBUS.MB_MASTER.bFUNCTION_CODE:=16#03;
			MODBUS.MB_MASTER.wREAD_ADDRESS:=16#0D;
			MODBUS.MB_MASTER.wREAD_QUANTITY:=16#1;
			MODBUS.MB_Start:=TRUE;
			sta:=LQI_REQUEST;
		END_IF

	LQI_REQUEST:	(* Link quality *)
		IF NOT MODBUS.MB_Start THEN
			IF MODBUS.MB_MASTER.wERROR<>MB_NO_ERROR THEN
				sta:=ERROR_STATE;
			ELSE
				(*NodeStatus	:=	MODBUS.MB_READBUF[0];*)

				MODBUS.ID:=ID;
				MODBUS.MB_MASTER.bUNIT_ID := Address;
				MODBUS.MB_MASTER.bFUNCTION_CODE:=16#03;
				MODBUS.MB_MASTER.wREAD_ADDRESS:=16#01;
				MODBUS.MB_MASTER.wREAD_QUANTITY:=16#1;
				MODBUS.MB_Start:=TRUE;

				sta:=MEAS_REQUEST;
			END_IF
		END_IF

	MEAS_REQUEST:	(* Measurements *)
		IF NOT MODBUS.MB_Start THEN
			IF MODBUS.MB_MASTER.wERROR<>MB_NO_ERROR THEN
				sta:=ERROR_STATE;
			ELSE

				OUT_LQI	:=	WORD_TO_BYTE(MODBUS.MB_READBUF[0]);

				MODBUS.ID:=ID;
				MODBUS.MB_MASTER.bUNIT_ID := Address;
				MODBUS.MB_MASTER.bFUNCTION_CODE:=16#03;
				MODBUS.MB_MASTER.wREAD_ADDRESS:=16#14;
				MODBUS.MB_MASTER.wREAD_QUANTITY:=16#5;
				MODBUS.MB_Start:=TRUE;

				sta:=END_READ;
			END_IF
		END_IF

	END_READ:	IF NOT MODBUS.MB_Start THEN
			IF MODBUS.MB_MASTER.wERROR<>MB_NO_ERROR THEN
				sta:=ERROR_STATE;
			ELSE
				OUT_TEMP	:=	WORD_TO_INT(MODBUS.MB_READBUF[0]);
				OUT_HYGRO	:=	WORD_TO_INT(MODBUS.MB_READBUF[1]);
				OUT_LUX		:=	WORD_TO_INT(MODBUS.MB_READBUF[2]);
				OUT_VBATT	:=	WORD_TO_INT(MODBUS.MB_READBUF[3]);
				sta:=WAIT_STATE;
				MODBUS.MB_Lock:=FALSE;
			END_IF
		END_IF

	ERROR_STATE:
			MODBUS.MB_Lock:=FALSE;
			(* Retries *)
			retry:=retry+1;
			IF retry>3 THEN
				retry:=0;
				IF Status_Log<>2 THEN
					LogEv(EL_Alarm,EO_ZTHL,ID,4,'');
				END_IF
				Status_Log:=2;
				Status_Vis:=COLOR_RED;
			END_IF
			sta:=WAIT_STATE;

ELSE
			sta:=WAIT_STATE;
END_CASE

(* Check Status *)
(*
IF NodeStatus <> OldNodeStatus THEN
	IF NodeStatus = 3 THEN
		LogEv(EL_Alarm,EO_ZTHL,ID,3,'');
		Status_Log:=2;
	ELSE
		Status_Log:=0;
	END_IF

	OldNodeStatus := NodeStatus;
END_IF*)

(* Check Link quality *)
IF OUT_LQI > LQI_Threshold THEN
	fLQI := TRUE;
	ERR := TRUE;
ELSE
	fLQI := FALSE;
	ERR := FALSE;
END_IF

Quality(IN:=fLQI);

IF Quality.EVL THEN
	LogEv(SEL(OUT_LQI<>0,EL_Alarm,EL_Wrn),EO_ZTHL,ID,SEL(OUT_LQI<>0,7,2),WORD_TO_STRING(OUT_LQI));
	Status_Log := SEL(OUT_LQI<>0,2,1);
	StatusOK := StatusOK + 1;
END_IF

IF Quality.EVH THEN StatusOK := SEL(StatusOK=0, StatusOK-1, 0); END_IF

(* If probe (node) is present proceed checking other warnings, otherwise don't transmit anything *)
IF OUT_LQI <> 0 THEN

	(* Check battery voltage *)
	IF OUT_VBATT < LowBattVoltage THEN fBatt := TRUE;
	ELSE fBatt := FALSE;
	END_IF
	
	Battery(IN:=fBatt);
	
	IF Battery.EVH THEN
		LogEv(EL_Wrn,EO_ZTHL,ID,6,'');
		StatusOK := StatusOK + 1;
	END_IF

	IF Battery.EVL THEN StatusOK := SEL(StatusOK=0, StatusOK-1, 0); END_IF

	(* Check Node temperature *)
	IF OUT_TEMP < Tmin OR OUT_TEMP > Tmax THEN
		fTemp := TRUE;
		ERR := TRUE;
	ELSE
		fTemp := FALSE;
		ERR := FALSE;
	END_IF

	Temperature(IN:=fTemp);

	IF Temperature.EVH THEN
		LogEv(EL_Wrn,EO_ZTHL,ID,5,INT_TO_STRING(OUT_TEMP));
		Status_Log := 1;
		StatusOK := StatusOK + 1;
	END_IF

	IF Temperature.EVL THEN StatusOK := SEL(StatusOK=0, StatusOK-1, 0); END_IF

END_IF

Alarm(IN:=(StatusOK=0));

IF Alarm.EVH THEN
	Status_Log := 0;
	LogEv(EL_Log,EO_ZTHL,ID,1,'');
END_IF

IF Status_Log = 2 THEN Status_Vis := COLOR_RED;
ELSIF Status_Log = 1 THEN Status_Vis := COLOR_YELLOW;
ELSE Status_Vis := COLOR_GREEN;
END_IF
END_FUNCTION_BLOCK
ACTION AddLogData:
Logger.s1:=INSERT('&ZTHL=',BYTE_TO_STRING(ID),5);
IF ID<10 THEN Logger.s1:=INSERT(Logger.s1,'0',5); END_IF

Logger.s1:=CONCAT(Logger.s1,BYTE_TO_STRING(OUT_LQI));			Logger.s1:=CONCAT(Logger.s1,';');
Logger.s1:=CONCAT(Logger.s1,INT_TO_STRING(OUT_TEMP ));			Logger.s1:=CONCAT(Logger.s1,';');
Logger.s1:=CONCAT(Logger.s1,INT_TO_STRING(OUT_HYGRO ));			Logger.s1:=CONCAT(Logger.s1,';');
Logger.s1:=CONCAT(Logger.s1,INT_TO_STRING(OUT_LUX));			Logger.s1:=CONCAT(Logger.s1,';');
Logger.s1:=CONCAT(Logger.s1,INT_TO_STRING(OUT_VBATT));			Logger.s1:=CONCAT(Logger.s1,';');

Logger.s1:=CONCAT(Logger.s1,BYTE_TO_STRING(Status_Log));
ADDSTRING(ADR(Logger.TData), ADR(Logger.s1), Logger.TLen);
END_ACTION

(* POU Utils Functions/PLANT_STATUS, ST *)
FUNCTION_BLOCK PLANT_STATUS
VAR_INPUT
	obj_Status		:	WORD;
END_VAR
VAR_OUTPUT
END_VAR
VAR
	PLANT_STATUS	:	WORD;

	Pwm				:	TON := (PT:=T#1s);
END_VAR
CASE plant_Status OF

	0:	(* Plant OK - Everything works well *)
		Pwm(IN:=FALSE);							(* Stop timer if running *)
		LAMP_AL := FALSE;						(* Keep the lamp switched off *)

	1:	(* Plant in warning *)
		Pwm(IN:= NOT(Pwm.Q));

		IF Pwm.Q THEN
			LAMP_AL := NOT LAMP_AL;				(* Toggle output *)
		END_IF

	2:	(* Plant in alarm *)
		Pwm(IN:=FALSE);							(* Stop timer if running *)
		LAMP_AL	:= TRUE;						(* Keep the lamp switched on *)

END_CASE

plant_Status := 0;		(* Reset plant status *)
END_FUNCTION_BLOCK
ACTION UpdateStatus:
IF plant_Status = 2 THEN

	RETURN;					(* If plant already in alarm condition do nothing *)

ELSE

		IF obj_Status <> 0 THEN
			plant_Status := obj_Status;			(* If plant in warning/normal condition and current object in alarm, update plant status *)
		END_IF
END_IF
END_ACTION

(* POU PLC_WDT, ST *)
FUNCTION PLC_WDT: DWORD VAR_INPUT dwEvent: DWORD; dwFilter: DWORD; dwOwner: DWORD; END_VAR
LogEv(EL_AlarmStop,EO_SYS,1,10,'Watchdog');
END_FUNCTION

(* POU Utils Functions/RAW16TOHEXSTR, ST *)
FUNCTION RAW16TOHEXSTR : STRING(128)
VAR_INPUT
	pData: POINTER TO BYTE;
	DataLen: BYTE;
END_VAR
VAR
	pt: POINTER TO BYTE;
	xl: BYTE;
END_VAR
pt:=ADR(RAW16TOHEXSTR);
xl:=0;

WHILE DataLen>0 AND xl<120 DO

	pData:=pData+1;

	pt^ := (pData^ / 16#10) + 48 + (((pData^ / 16#10)/10)*7);
	pt:=pt+1;
	pt^ := (pData^ AND 16#0F)  + 48 + (((pData^ AND 16#0F)/10)*7);
	pt:=pt+1;

	pData:=pData-1;

	pt^ := (pData^ / 16#10) + 48 + (((pData^ / 16#10)/10)*7);
	pt:=pt+1;
	pt^ := (pData^ AND 16#0F)  + 48 + (((pData^ AND 16#0F)/10)*7);
	pt:=pt+1;

	xl:=xl+4;

	DataLen:=DataLen-2;
	pData:=pData+2;

END_WHILE

pt^:=0;
END_FUNCTION

(* POU Utils/RTC_Update, ST *)
FUNCTION RTC_Update : BOOL
VAR
	T: DT;
	TS: STRING;
	TS2: STRING;
	Hour: BYTE;
	Minute: BYTE;
END_VAR
(* Get RTC time *)
T:=SysRtcGetTime(TRUE);
Sys.Time_CT_DT:=T;
(* Calculate variables *)
TS:=DT_TO_STRING(T);
Sys.Time_LogString:=DELETE(STR:=TS, LEN:=3, POS:=1);
TS2:=MID(STR:=TS, LEN:=4, POS:= 4); Sys.Time_Year 	:=STRING_TO_WORD(TS2);
TS2:=MID(STR:=TS, LEN:=2, POS:= 9); Sys.Time_Month	:=STRING_TO_BYTE(TS2);
TS2:=MID(STR:=TS, LEN:=2, POS:=12); Sys.Time_Day  	:=STRING_TO_BYTE(TS2);
Sys.Time_CT_Day:=(32*(Sys.Time_Month-1)+Sys.Time_Day-1);
TS2:=MID(STR:=TS, LEN:=2, POS:=15); Hour			:=STRING_TO_BYTE(TS2);
TS2:=MID(STR:=TS, LEN:=2, POS:=18); Minute		 	:=STRING_TO_BYTE(TS2);
Sys.Time_CT_Quarter:=Hour*4+(Minute/15);
END_FUNCTION

(* Visualisation PLC_VISU
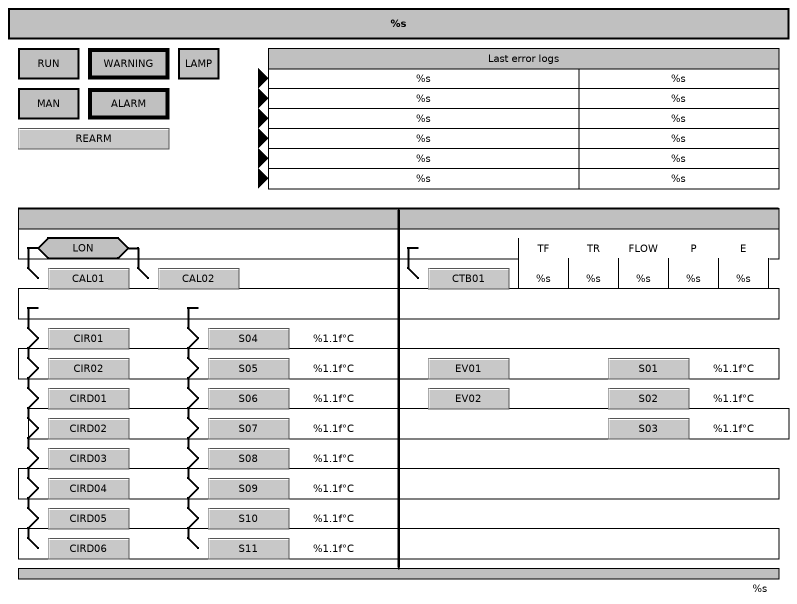
rectangle at (10,10)-(791,41): text "%s"; shows .Plant_NAME
rectangle at (530,580)-(771,601): text "%s"; shows Sys.Time_LogString
rounded rectangle at (20,50)-(81,81): text "RUN"; alarm colour if NOT Mode_Manual; runs INTERN ASSIGN Mode_Manual:=(FALSE)
rounded rectangle at (20,90)-(81,121): text "MAN"; alarm colour if Mode_Manual; runs INTERN ASSIGN Mode_Manual:=(TRUE)
rectangle at (580,70)-(781,91): text "%s"; shows Sys.LastLogs_Msg[0]
polygon at (260,170)-(270,190): invisible if Sys.LastLogs_Idx<>0
rectangle at (580,90)-(781,111): text "%s"; shows Sys.LastLogs_Msg[1]
polygon at (260,70)-(270,90): invisible if Sys.LastLogs_Idx<>1
rectangle at (580,110)-(781,131): text "%s"; shows Sys.LastLogs_Msg[2]
polygon at (260,90)-(270,110): invisible if Sys.LastLogs_Idx<>2
rectangle at (580,130)-(781,151): text "%s"; shows Sys.LastLogs_Msg[3]
polygon at (260,110)-(270,130): invisible if Sys.LastLogs_Idx<>3
rectangle at (580,150)-(781,171): text "%s"; shows Sys.LastLogs_Msg[4]
polygon at (260,130)-(270,150): invisible if Sys.LastLogs_Idx<>4
rectangle at (580,170)-(781,191): text "%s"; shows Sys.LastLogs_Msg[5]
polygon at (260,150)-(270,170): invisible if Sys.LastLogs_Idx<>5
rectangle at (270,70)-(581,91): text "%s"; shows Sys.LastLogs_Dat[0]
rectangle at (270,90)-(581,111): text "%s"; shows Sys.LastLogs_Dat[1]
rectangle at (270,110)-(581,131): text "%s"; shows Sys.LastLogs_Dat[2]
rectangle at (270,130)-(581,151): text "%s"; shows Sys.LastLogs_Dat[3]
rectangle at (270,150)-(581,171): text "%s"; shows Sys.LastLogs_Dat[4]
rectangle at (270,170)-(581,191): text "%s"; shows Sys.LastLogs_Dat[5]
rectangle at (90,90)-(171,121): text "ALARM"; alarm colour if Sys.Alarm; runs INTERN ASSIGN Mode_Manual:=(FALSE)
rectangle at (90,50)-(171,81): text "WARNING"; alarm colour if Sys.Warning; runs INTERN ASSIGN Mode_Manual:=(TRUE)
button at (20,130)-(171,151): text "REARM"; runs INTERN ASSIGN Sys.Alarm:=(FALSE);INTERN ASSIGN Sys.Warning:=(FALSE)
button at (430,270)-(511,291): text "CTB01"
rectangle at (270,50)-(781,71): text "Last error logs"
rectangle at (520,240)-(571,261): text "TF"
rectangle at (620,240)-(671,261): text "FLOW"
rectangle at (670,240)-(721,261): text "P"
rectangle at (720,240)-(771,261): text "E"
rectangle at (570,240)-(621,261): text "TR"
rectangle at (520,270)-(571,291): text "%s"; shows .CTB01.M1.utFTemp.Value
rectangle at (620,270)-(671,291): text "%s"; shows .CTB01.M1.utFlow.Value
rectangle at (670,270)-(721,291): text "%s"; shows CTB01.M1.utPower.Value
rectangle at (720,270)-(771,291): text "%s"; shows CTB01.M1.utEnergy.Value
rectangle at (570,270)-(621,291): text "%s"; shows .CTB01.M1.utRTemp.Value
button at (50,390)-(131,411): text "CIRD01"
button at (50,420)-(131,441): text "CIRD02"
button at (50,450)-(131,471): text "CIRD03"
button at (50,330)-(131,351): text "CIR01"
button at (50,480)-(131,501): text "CIRD04"
button at (50,360)-(131,381): text "CIR02"
button at (610,360)-(691,381): text "S01"; opens Vis_VRD02
button at (610,390)-(691,411): text "S02"; opens Vis_VRD02
button at (610,420)-(691,441): text "S03"; opens Vis_VRD02
button at (210,330)-(291,351): text "S04"; opens Vis_VRD02
button at (210,360)-(291,381): text "S05"; opens Vis_VRD02
button at (210,390)-(291,411): text "S06"; opens Vis_VRD02
button at (210,420)-(291,441): text "S07"; opens Vis_VRD02
button at (210,450)-(291,471): text "S08"; opens Vis_VRD02
button at (210,480)-(291,501): text "S09"; opens Vis_VRD02
button at (210,510)-(291,531): text "S10"; opens Vis_VRD02
button at (210,540)-(291,561): text "S11"; opens Vis_VRD02
rectangle at (690,360)-(781,381): text "%1.1f°C"; shows INT_TO_REAL(.TPV01.IN)/10
rectangle at (690,390)-(781,411): text "%1.1f°C"; shows INT_TO_REAL(.TPV02.IN)/10
rectangle at (690,420)-(781,441): text "%1.1f°C"; shows INT_TO_REAL(.TPV03.IN)/10
rectangle at (290,330)-(381,351): text "%1.1f°C"; shows INT_TO_REAL(ZTHL04.OUT_TEMP)/10
rectangle at (290,360)-(381,381): text "%1.1f°C"; shows INT_TO_REAL(ZTHL05.OUT_TEMP)/10
rectangle at (290,390)-(381,411): text "%1.1f°C"; shows INT_TO_REAL(.ZTHL06.OUT_TEMP)/10
rectangle at (290,420)-(381,441): text "%1.1f°C"; shows INT_TO_REAL(ZTHL07.OUT_TEMP)/10
rectangle at (290,450)-(381,471): text "%1.1f°C"; shows INT_TO_REAL(ZTHL08.OUT_TEMP)/10
rectangle at (290,480)-(381,501): text "%1.1f°C"; shows INT_TO_REAL(ZTHL09.OUT_TEMP)/10
rectangle at (290,510)-(381,531): text "%1.1f°C"; shows INT_TO_REAL(ZTHL10.OUT_TEMP)/10
rectangle at (290,540)-(381,561): text "%1.1f°C"; shows INT_TO_REAL(ZTHL11.OUT_TEMP)/10
button at (50,270)-(131,291): text "CAL01"; opens Vis_CAL01
polygon at (40,240)-(130,260): text "LON"
button at (160,270)-(241,291): text "CAL02"; opens Vis_CAL01
button at (50,510)-(131,531): text "CIRD05"
button at (50,540)-(131,561): text "CIRD06"
button at (430,360)-(511,381): text "EV01"; opens Vis_VRD02
button at (430,390)-(511,411): text "EV02"; opens Vis_VRD02
rounded rectangle at (180,50)-(221,81): text "LAMP"; alarm colour if LAMP_AL
35 more shapes without text or variables
27 elements of other kinds (tables, trends, ...) not read
*)

(* Visualisation VIS_CAL01
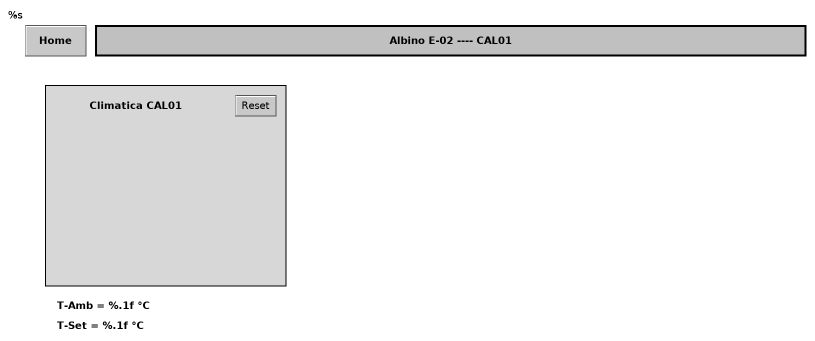
rectangle at (40,300)-(181,321): text "T-Set = %.1f °C"; shows INT_TO_REAL(CAL01.CFD_SetPoint.iSnvtTempP)/100
rectangle at (0,0)-(0,0): text "%s"; shows CAL01_Clima.Points[INDEX].X; invisible if INDEX>4; editable
rectangle at (0,0)-(0,0): text "%s"; shows CAL01_Clima.Points[INDEX].Y; invisible if INDEX>4; editable
rectangle at (40,280)-(181,301): text "T-Amb = %.1f °C"; shows INT_TO_REAL(.T_AMB)/10; alarm colour if T_AMB>2000
rectangle at (40,80)-(201,101): text "Climatica CAL01"
button at (220,80)-(261,101): text "Reset"; runs INTERN ASSIGN CAL01_Clima.InitOK:=(FALSE)
rectangle at (80,10)-(791,41): text "Albino E-02 ---- CAL01"
button at (10,10)-(71,41): text "Home"; opens PLC_VISU
1 more shapes without text or variables
*)

(* Visualisation VIS_CHONOEDITOR
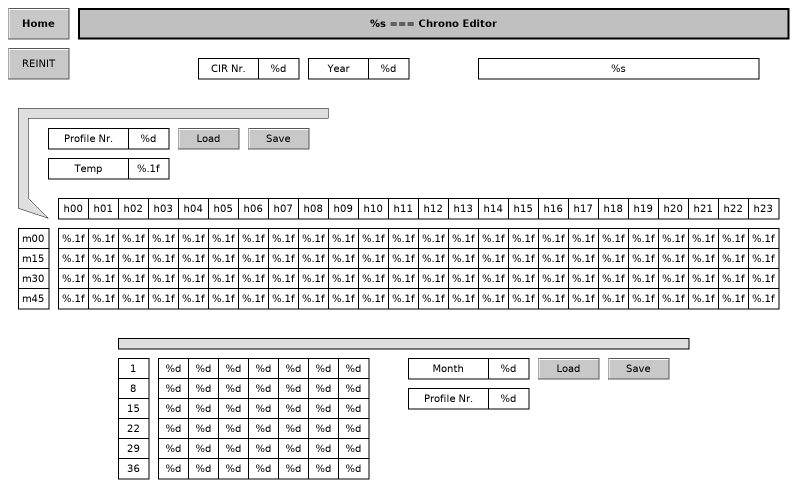
rectangle at (200,60)-(261,81): text "CIR Nr."
rectangle at (260,60)-(301,81): text "%d"; shows CronEd.CN_Sel; alarm colour if CronEd.CN_Sel<>CronEd.CN_Act; editable 1..7
rectangle at (50,130)-(131,151): text "Profile Nr."
rectangle at (130,130)-(171,151): text "%d"; shows CronEd.PR_Sel; alarm colour if CronEd.PR_Sel<>CronEd.PR_Act; editable 1..10
rectangle at (50,160)-(131,181): text "Temp"
rectangle at (130,160)-(171,181): text "%.1f"; shows CronEd.PR_TT; editable
button at (180,130)-(241,151): text "Load"; toggles CronEd.PR_Load
button at (250,130)-(311,151): text "Save"; toggles CronEd.PR_Save
rectangle at (20,230)-(51,251): text "m00"
rectangle at (20,250)-(51,271): text "m15"
rectangle at (20,270)-(51,291): text "m30"
rectangle at (20,290)-(51,311): text "m45"
rectangle at (80,10)-(791,41): text "%s === Chrono Editor"; shows .Plant_NAME
button at (10,10)-(71,41): text "Home"; opens PLC_VISU
rounded rectangle at (60,230)-(91,251): text "%.1f"; shows WORD_TO_REAL(CronEd.PR.Setpoint[0])/10; runs INTERN ASSIGN CronEd.PR.Setpoint[0]:=(REAL_TO_WORD(CronEd.PR_TT*10))
rounded rectangle at (60,250)-(91,271): text "%.1f"; shows WORD_TO_REAL(CronEd.PR.Setpoint[1])/10; runs INTERN ASSIGN CronEd.PR.Setpoint[1]:=(REAL_TO_WORD(CronEd.PR_TT*10))
rounded rectangle at (60,270)-(91,291): text "%.1f"; shows WORD_TO_REAL(CronEd.PR.Setpoint[2])/10; runs INTERN ASSIGN CronEd.PR.Setpoint[2]:=(REAL_TO_WORD(CronEd.PR_TT*10))
rounded rectangle at (60,290)-(91,311): text "%.1f"; shows WORD_TO_REAL(CronEd.PR.Setpoint[3])/10; runs INTERN ASSIGN CronEd.PR.Setpoint[3]:=(REAL_TO_WORD(CronEd.PR_TT*10))
rectangle at (60,200)-(91,221): text "h00"; runs INTERN ASSIGN CronEd.PR.Setpoint[0]:=(REAL_TO_WORD(CronEd.PR_TT*10));INTERN ASSIGN CronEd.PR.Setpoint[1]:=(REAL_TO_WORD(CronEd.PR_TT*10));INTERN ASSIGN CronEd.PR.Setpoint[2]:=(REAL_TO_WORD(CronEd.PR_TT*10));INTERN ASSIGN CronEd.PR.Setpoint[3]:=(REAL_TO_WORD(CronEd.PR_TT*10))
rounded rectangle at (90,230)-(121,251): text "%.1f"; shows WORD_TO_REAL(CronEd.PR.Setpoint[4])/10; runs INTERN ASSIGN CronEd.PR.Setpoint[4]:=(REAL_TO_WORD(CronEd.PR_TT*10))
rounded rectangle at (90,250)-(121,271): text "%.1f"; shows WORD_TO_REAL(CronEd.PR.Setpoint[5])/10; runs INTERN ASSIGN CronEd.PR.Setpoint[5]:=(REAL_TO_WORD(CronEd.PR_TT*10))
rounded rectangle at (90,270)-(121,291): text "%.1f"; shows WORD_TO_REAL(CronEd.PR.Setpoint[6])/10; runs INTERN ASSIGN CronEd.PR.Setpoint[6]:=(REAL_TO_WORD(CronEd.PR_TT*10))
rounded rectangle at (90,290)-(121,311): text "%.1f"; shows WORD_TO_REAL(CronEd.PR.Setpoint[7])/10; runs INTERN ASSIGN CronEd.PR.Setpoint[7]:=(REAL_TO_WORD(CronEd.PR_TT*10))
rectangle at (90,200)-(121,221): text "h01"; runs INTERN ASSIGN CronEd.PR.Setpoint[4]:=(REAL_TO_WORD(CronEd.PR_TT*10));INTERN ASSIGN CronEd.PR.Setpoint[5]:=(REAL_TO_WORD(CronEd.PR_TT*10));INTERN ASSIGN CronEd.PR.Setpoint[6]:=(REAL_TO_WORD(CronEd.PR_TT*10));INTERN ASSIGN CronEd.PR.Setpoint[7]:=(REAL_TO_WORD(CronEd.PR_TT*10))
rounded rectangle at (120,230)-(151,251): text "%.1f"; shows WORD_TO_REAL(CronEd.PR.Setpoint[8])/10; runs INTERN ASSIGN CronEd.PR.Setpoint[8]:=(REAL_TO_WORD(CronEd.PR_TT*10))
rounded rectangle at (120,250)-(151,271): text "%.1f"; shows WORD_TO_REAL(CronEd.PR.Setpoint[9])/10; runs INTERN ASSIGN CronEd.PR.Setpoint[9]:=(REAL_TO_WORD(CronEd.PR_TT*10))
rounded rectangle at (120,270)-(151,291): text "%.1f"; shows WORD_TO_REAL(CronEd.PR.Setpoint[10])/10; runs INTERN ASSIGN CronEd.PR.Setpoint[10]:=(REAL_TO_WORD(CronEd.PR_TT*10))
rounded rectangle at (120,290)-(151,311): text "%.1f"; shows WORD_TO_REAL(CronEd.PR.Setpoint[11])/10; runs INTERN ASSIGN CronEd.PR.Setpoint[11]:=(REAL_TO_WORD(CronEd.PR_TT*10))
rectangle at (120,200)-(151,221): text "h02"; runs INTERN ASSIGN CronEd.PR.Setpoint[8]:=(REAL_TO_WORD(CronEd.PR_TT*10));INTERN ASSIGN CronEd.PR.Setpoint[9]:=(REAL_TO_WORD(CronEd.PR_TT*10));INTERN ASSIGN CronEd.PR.Setpoint[10]:=(REAL_TO_WORD(CronEd.PR_TT*10));INTERN ASSIGN CronEd.PR.Setpoint[11]:=(REAL_TO_WORD(CronEd.PR_TT*10))
rounded rectangle at (150,230)-(181,251): text "%.1f"; shows WORD_TO_REAL(CronEd.PR.Setpoint[12])/10; runs INTERN ASSIGN CronEd.PR.Setpoint[12]:=(REAL_TO_WORD(CronEd.PR_TT*10))
rounded rectangle at (150,250)-(181,271): text "%.1f"; shows WORD_TO_REAL(CronEd.PR.Setpoint[13])/10; runs INTERN ASSIGN CronEd.PR.Setpoint[13]:=(REAL_TO_WORD(CronEd.PR_TT*10))
rounded rectangle at (150,270)-(181,291): text "%.1f"; shows WORD_TO_REAL(CronEd.PR.Setpoint[14])/10; runs INTERN ASSIGN CronEd.PR.Setpoint[14]:=(REAL_TO_WORD(CronEd.PR_TT*10))
rounded rectangle at (150,290)-(181,311): text "%.1f"; shows WORD_TO_REAL(CronEd.PR.Setpoint[15])/10; runs INTERN ASSIGN CronEd.PR.Setpoint[15]:=(REAL_TO_WORD(CronEd.PR_TT*10))
rectangle at (150,200)-(181,221): text "h03"; runs INTERN ASSIGN CronEd.PR.Setpoint[15]:=(REAL_TO_WORD(CronEd.PR_TT*10));INTERN ASSIGN CronEd.PR.Setpoint[14]:=(REAL_TO_WORD(CronEd.PR_TT*10));INTERN ASSIGN CronEd.PR.Setpoint[13]:=(REAL_TO_WORD(CronEd.PR_TT*10));INTERN ASSIGN CronEd.PR.Setpoint[12]:=(REAL_TO_WORD(CronEd.PR_TT*10))
rounded rectangle at (180,230)-(211,251): text "%.1f"; shows WORD_TO_REAL(CronEd.PR.Setpoint[16])/10; runs INTERN ASSIGN CronEd.PR.Setpoint[16]:=(REAL_TO_WORD(CronEd.PR_TT*10))
rounded rectangle at (180,250)-(211,271): text "%.1f"; shows WORD_TO_REAL(CronEd.PR.Setpoint[17])/10; runs INTERN ASSIGN CronEd.PR.Setpoint[17]:=(REAL_TO_WORD(CronEd.PR_TT*10))
rounded rectangle at (180,270)-(211,291): text "%.1f"; shows WORD_TO_REAL(CronEd.PR.Setpoint[18])/10; runs INTERN ASSIGN CronEd.PR.Setpoint[18]:=(REAL_TO_WORD(CronEd.PR_TT*10))
rounded rectangle at (180,290)-(211,311): text "%.1f"; shows WORD_TO_REAL(CronEd.PR.Setpoint[19])/10; runs INTERN ASSIGN CronEd.PR.Setpoint[19]:=(REAL_TO_WORD(CronEd.PR_TT*10))
rectangle at (180,200)-(211,221): text "h04"; runs INTERN ASSIGN CronEd.PR.Setpoint[19]:=(REAL_TO_WORD(CronEd.PR_TT*10));INTERN ASSIGN CronEd.PR.Setpoint[18]:=(REAL_TO_WORD(CronEd.PR_TT*10));INTERN ASSIGN CronEd.PR.Setpoint[17]:=(REAL_TO_WORD(CronEd.PR_TT*10));INTERN ASSIGN CronEd.PR.Setpoint[16]:=(REAL_TO_WORD(CronEd.PR_TT*10))
rounded rectangle at (210,230)-(241,251): text "%.1f"; shows WORD_TO_REAL(CronEd.PR.Setpoint[20])/10; runs INTERN ASSIGN CronEd.PR.Setpoint[20]:=(REAL_TO_WORD(CronEd.PR_TT*10))
rounded rectangle at (210,250)-(241,271): text "%.1f"; shows WORD_TO_REAL(CronEd.PR.Setpoint[21])/10; runs INTERN ASSIGN CronEd.PR.Setpoint[21]:=(REAL_TO_WORD(CronEd.PR_TT*10))
rounded rectangle at (210,270)-(241,291): text "%.1f"; shows WORD_TO_REAL(CronEd.PR.Setpoint[22])/10; runs INTERN ASSIGN CronEd.PR.Setpoint[22]:=(REAL_TO_WORD(CronEd.PR_TT*10))
rounded rectangle at (210,290)-(241,311): text "%.1f"; shows WORD_TO_REAL(CronEd.PR.Setpoint[23])/10; runs INTERN ASSIGN CronEd.PR.Setpoint[23]:=(REAL_TO_WORD(CronEd.PR_TT*10))
rectangle at (210,200)-(241,221): text "h05"; runs INTERN ASSIGN CronEd.PR.Setpoint[23]:=(REAL_TO_WORD(CronEd.PR_TT*10));INTERN ASSIGN CronEd.PR.Setpoint[22]:=(REAL_TO_WORD(CronEd.PR_TT*10));INTERN ASSIGN CronEd.PR.Setpoint[21]:=(REAL_TO_WORD(CronEd.PR_TT*10));INTERN ASSIGN CronEd.PR.Setpoint[20]:=(REAL_TO_WORD(CronEd.PR_TT*10))
rounded rectangle at (240,230)-(271,251): text "%.1f"; shows WORD_TO_REAL(CronEd.PR.Setpoint[24])/10; runs INTERN ASSIGN CronEd.PR.Setpoint[24]:=(REAL_TO_WORD(CronEd.PR_TT*10))
rounded rectangle at (240,250)-(271,271): text "%.1f"; shows WORD_TO_REAL(CronEd.PR.Setpoint[25])/10; runs INTERN ASSIGN CronEd.PR.Setpoint[25]:=(REAL_TO_WORD(CronEd.PR_TT*10))
rounded rectangle at (240,270)-(271,291): text "%.1f"; shows WORD_TO_REAL(CronEd.PR.Setpoint[26])/10; runs INTERN ASSIGN CronEd.PR.Setpoint[26]:=(REAL_TO_WORD(CronEd.PR_TT*10))
rounded rectangle at (240,290)-(271,311): text "%.1f"; shows WORD_TO_REAL(CronEd.PR.Setpoint[27])/10; runs INTERN ASSIGN CronEd.PR.Setpoint[27]:=(REAL_TO_WORD(CronEd.PR_TT*10))
rectangle at (240,200)-(271,221): text "h06"; runs INTERN ASSIGN CronEd.PR.Setpoint[27]:=(REAL_TO_WORD(CronEd.PR_TT*10));INTERN ASSIGN CronEd.PR.Setpoint[26]:=(REAL_TO_WORD(CronEd.PR_TT*10));INTERN ASSIGN CronEd.PR.Setpoint[25]:=(REAL_TO_WORD(CronEd.PR_TT*10));INTERN ASSIGN CronEd.PR.Setpoint[24]:=(REAL_TO_WORD(CronEd.PR_TT*10))
rounded rectangle at (270,230)-(301,251): text "%.1f"; shows WORD_TO_REAL(CronEd.PR.Setpoint[28])/10; runs INTERN ASSIGN CronEd.PR.Setpoint[28]:=(REAL_TO_WORD(CronEd.PR_TT*10))
rounded rectangle at (270,250)-(301,271): text "%.1f"; shows WORD_TO_REAL(CronEd.PR.Setpoint[29])/10; runs INTERN ASSIGN CronEd.PR.Setpoint[29]:=(REAL_TO_WORD(CronEd.PR_TT*10))
rounded rectangle at (270,270)-(301,291): text "%.1f"; shows WORD_TO_REAL(CronEd.PR.Setpoint[30])/10; runs INTERN ASSIGN CronEd.PR.Setpoint[30]:=(REAL_TO_WORD(CronEd.PR_TT*10))
rounded rectangle at (270,290)-(301,311): text "%.1f"; shows WORD_TO_REAL(CronEd.PR.Setpoint[31])/10; runs INTERN ASSIGN CronEd.PR.Setpoint[31]:=(REAL_TO_WORD(CronEd.PR_TT*10))
rectangle at (270,200)-(301,221): text "h07"; runs INTERN ASSIGN CronEd.PR.Setpoint[31]:=(REAL_TO_WORD(CronEd.PR_TT*10));INTERN ASSIGN CronEd.PR.Setpoint[30]:=(REAL_TO_WORD(CronEd.PR_TT*10));INTERN ASSIGN CronEd.PR.Setpoint[29]:=(REAL_TO_WORD(CronEd.PR_TT*10));INTERN ASSIGN CronEd.PR.Setpoint[28]:=(REAL_TO_WORD(CronEd.PR_TT*10))
rounded rectangle at (300,230)-(331,251): text "%.1f"; shows WORD_TO_REAL(CronEd.PR.Setpoint[32])/10; runs INTERN ASSIGN CronEd.PR.Setpoint[32]:=(REAL_TO_WORD(CronEd.PR_TT*10))
rounded rectangle at (300,250)-(331,271): text "%.1f"; shows WORD_TO_REAL(CronEd.PR.Setpoint[33])/10; runs INTERN ASSIGN CronEd.PR.Setpoint[33]:=(REAL_TO_WORD(CronEd.PR_TT*10))
rounded rectangle at (300,270)-(331,291): text "%.1f"; shows WORD_TO_REAL(CronEd.PR.Setpoint[34])/10; runs INTERN ASSIGN CronEd.PR.Setpoint[34]:=(REAL_TO_WORD(CronEd.PR_TT*10))
rounded rectangle at (300,290)-(331,311): text "%.1f"; shows WORD_TO_REAL(CronEd.PR.Setpoint[35])/10; runs INTERN ASSIGN CronEd.PR.Setpoint[35]:=(REAL_TO_WORD(CronEd.PR_TT*10))
rectangle at (300,200)-(331,221): text "h08"; runs INTERN ASSIGN CronEd.PR.Setpoint[35]:=(REAL_TO_WORD(CronEd.PR_TT*10));INTERN ASSIGN CronEd.PR.Setpoint[34]:=(REAL_TO_WORD(CronEd.PR_TT*10));INTERN ASSIGN CronEd.PR.Setpoint[33]:=(REAL_TO_WORD(CronEd.PR_TT*10));INTERN ASSIGN CronEd.PR.Setpoint[32]:=(REAL_TO_WORD(CronEd.PR_TT*10))
rounded rectangle at (330,230)-(361,251): text "%.1f"; shows WORD_TO_REAL(CronEd.PR.Setpoint[36])/10; runs INTERN ASSIGN CronEd.PR.Setpoint[36]:=(REAL_TO_WORD(CronEd.PR_TT*10))
rounded rectangle at (330,250)-(361,271): text "%.1f"; shows WORD_TO_REAL(CronEd.PR.Setpoint[37])/10; runs INTERN ASSIGN CronEd.PR.Setpoint[37]:=(REAL_TO_WORD(CronEd.PR_TT*10))
rounded rectangle at (330,270)-(361,291): text "%.1f"; shows WORD_TO_REAL(CronEd.PR.Setpoint[38])/10; runs INTERN ASSIGN CronEd.PR.Setpoint[38]:=(REAL_TO_WORD(CronEd.PR_TT*10))
rounded rectangle at (330,290)-(361,311): text "%.1f"; shows WORD_TO_REAL(CronEd.PR.Setpoint[39])/10; runs INTERN ASSIGN CronEd.PR.Setpoint[39]:=(REAL_TO_WORD(CronEd.PR_TT*10))
rectangle at (330,200)-(361,221): text "h09"; runs INTERN ASSIGN CronEd.PR.Setpoint[39]:=(REAL_TO_WORD(CronEd.PR_TT*10));INTERN ASSIGN CronEd.PR.Setpoint[38]:=(REAL_TO_WORD(CronEd.PR_TT*10));INTERN ASSIGN CronEd.PR.Setpoint[37]:=(REAL_TO_WORD(CronEd.PR_TT*10));INTERN ASSIGN CronEd.PR.Setpoint[36]:=(REAL_TO_WORD(CronEd.PR_TT*10))
rounded rectangle at (360,230)-(391,251): text "%.1f"; shows WORD_TO_REAL(CronEd.PR.Setpoint[40])/10; runs INTERN ASSIGN CronEd.PR.Setpoint[40]:=(REAL_TO_WORD(CronEd.PR_TT*10))
rounded rectangle at (360,250)-(391,271): text "%.1f"; shows WORD_TO_REAL(CronEd.PR.Setpoint[41])/10; runs INTERN ASSIGN CronEd.PR.Setpoint[41]:=(REAL_TO_WORD(CronEd.PR_TT*10))
rounded rectangle at (360,270)-(391,291): text "%.1f"; shows WORD_TO_REAL(CronEd.PR.Setpoint[42])/10; runs INTERN ASSIGN CronEd.PR.Setpoint[42]:=(REAL_TO_WORD(CronEd.PR_TT*10))
rounded rectangle at (360,290)-(391,311): text "%.1f"; shows WORD_TO_REAL(CronEd.PR.Setpoint[43])/10; runs INTERN ASSIGN CronEd.PR.Setpoint[43]:=(REAL_TO_WORD(CronEd.PR_TT*10))
rectangle at (360,200)-(391,221): text "h10"; runs INTERN ASSIGN CronEd.PR.Setpoint[43]:=(REAL_TO_WORD(CronEd.PR_TT*10));INTERN ASSIGN CronEd.PR.Setpoint[42]:=(REAL_TO_WORD(CronEd.PR_TT*10));INTERN ASSIGN CronEd.PR.Setpoint[41]:=(REAL_TO_WORD(CronEd.PR_TT*10));INTERN ASSIGN CronEd.PR.Setpoint[40]:=(REAL_TO_WORD(CronEd.PR_TT*10))
rounded rectangle at (390,230)-(421,251): text "%.1f"; shows WORD_TO_REAL(CronEd.PR.Setpoint[44])/10; runs INTERN ASSIGN CronEd.PR.Setpoint[44]:=(REAL_TO_WORD(CronEd.PR_TT*10))
rounded rectangle at (390,250)-(421,271): text "%.1f"; shows WORD_TO_REAL(CronEd.PR.Setpoint[45])/10; runs INTERN ASSIGN CronEd.PR.Setpoint[45]:=(REAL_TO_WORD(CronEd.PR_TT*10))
rounded rectangle at (390,270)-(421,291): text "%.1f"; shows WORD_TO_REAL(CronEd.PR.Setpoint[46])/10; runs INTERN ASSIGN CronEd.PR.Setpoint[46]:=(REAL_TO_WORD(CronEd.PR_TT*10))
rounded rectangle at (390,290)-(421,311): text "%.1f"; shows WORD_TO_REAL(CronEd.PR.Setpoint[47])/10; runs INTERN ASSIGN CronEd.PR.Setpoint[47]:=(REAL_TO_WORD(CronEd.PR_TT*10))
rectangle at (390,200)-(421,221): text "h11"; runs INTERN ASSIGN CronEd.PR.Setpoint[47]:=(REAL_TO_WORD(CronEd.PR_TT*10));INTERN ASSIGN CronEd.PR.Setpoint[46]:=(REAL_TO_WORD(CronEd.PR_TT*10));INTERN ASSIGN CronEd.PR.Setpoint[45]:=(REAL_TO_WORD(CronEd.PR_TT*10));INTERN ASSIGN CronEd.PR.Setpoint[44]:=(REAL_TO_WORD(CronEd.PR_TT*10))
rounded rectangle at (420,230)-(451,251): text "%.1f"; shows WORD_TO_REAL(CronEd.PR.Setpoint[48])/10; runs INTERN ASSIGN CronEd.PR.Setpoint[48]:=(REAL_TO_WORD(CronEd.PR_TT*10))
rounded rectangle at (420,250)-(451,271): text "%.1f"; shows WORD_TO_REAL(CronEd.PR.Setpoint[49])/10; runs INTERN ASSIGN CronEd.PR.Setpoint[49]:=(REAL_TO_WORD(CronEd.PR_TT*10))
rounded rectangle at (420,270)-(451,291): text "%.1f"; shows WORD_TO_REAL(CronEd.PR.Setpoint[50])/10; runs INTERN ASSIGN CronEd.PR.Setpoint[50]:=(REAL_TO_WORD(CronEd.PR_TT*10))
rounded rectangle at (420,290)-(451,311): text "%.1f"; shows WORD_TO_REAL(CronEd.PR.Setpoint[51])/10; runs INTERN ASSIGN CronEd.PR.Setpoint[51]:=(REAL_TO_WORD(CronEd.PR_TT*10))
rectangle at (420,200)-(451,221): text "h12"; runs INTERN ASSIGN CronEd.PR.Setpoint[51]:=(REAL_TO_WORD(CronEd.PR_TT*10));INTERN ASSIGN CronEd.PR.Setpoint[50]:=(REAL_TO_WORD(CronEd.PR_TT*10));INTERN ASSIGN CronEd.PR.Setpoint[49]:=(REAL_TO_WORD(CronEd.PR_TT*10));INTERN ASSIGN CronEd.PR.Setpoint[48]:=(REAL_TO_WORD(CronEd.PR_TT*10))
rounded rectangle at (450,230)-(481,251): text "%.1f"; shows WORD_TO_REAL(CronEd.PR.Setpoint[52])/10; runs INTERN ASSIGN CronEd.PR.Setpoint[52]:=(REAL_TO_WORD(CronEd.PR_TT*10))
rounded rectangle at (450,250)-(481,271): text "%.1f"; shows WORD_TO_REAL(CronEd.PR.Setpoint[53])/10; runs INTERN ASSIGN CronEd.PR.Setpoint[53]:=(REAL_TO_WORD(CronEd.PR_TT*10))
rounded rectangle at (450,270)-(481,291): text "%.1f"; shows WORD_TO_REAL(CronEd.PR.Setpoint[54])/10; runs INTERN ASSIGN CronEd.PR.Setpoint[54]:=(REAL_TO_WORD(CronEd.PR_TT*10))
rounded rectangle at (450,290)-(481,311): text "%.1f"; shows WORD_TO_REAL(CronEd.PR.Setpoint[55])/10; runs INTERN ASSIGN CronEd.PR.Setpoint[55]:=(REAL_TO_WORD(CronEd.PR_TT*10))
rectangle at (450,200)-(481,221): text "h13"; runs INTERN ASSIGN CronEd.PR.Setpoint[55]:=(REAL_TO_WORD(CronEd.PR_TT*10));INTERN ASSIGN CronEd.PR.Setpoint[54]:=(REAL_TO_WORD(CronEd.PR_TT*10));INTERN ASSIGN CronEd.PR.Setpoint[53]:=(REAL_TO_WORD(CronEd.PR_TT*10));INTERN ASSIGN CronEd.PR.Setpoint[52]:=(REAL_TO_WORD(CronEd.PR_TT*10))
rounded rectangle at (480,230)-(511,251): text "%.1f"; shows WORD_TO_REAL(CronEd.PR.Setpoint[56])/10; runs INTERN ASSIGN CronEd.PR.Setpoint[56]:=(REAL_TO_WORD(CronEd.PR_TT*10))
rounded rectangle at (480,250)-(511,271): text "%.1f"; shows WORD_TO_REAL(CronEd.PR.Setpoint[57])/10; runs INTERN ASSIGN CronEd.PR.Setpoint[57]:=(REAL_TO_WORD(CronEd.PR_TT*10))
rounded rectangle at (480,270)-(511,291): text "%.1f"; shows WORD_TO_REAL(CronEd.PR.Setpoint[58])/10; runs INTERN ASSIGN CronEd.PR.Setpoint[58]:=(REAL_TO_WORD(CronEd.PR_TT*10))
rounded rectangle at (480,290)-(511,311): text "%.1f"; shows WORD_TO_REAL(CronEd.PR.Setpoint[59])/10; runs INTERN ASSIGN CronEd.PR.Setpoint[59]:=(REAL_TO_WORD(CronEd.PR_TT*10))
rectangle at (480,200)-(511,221): text "h14"; runs INTERN ASSIGN CronEd.PR.Setpoint[59]:=(REAL_TO_WORD(CronEd.PR_TT*10));INTERN ASSIGN CronEd.PR.Setpoint[58]:=(REAL_TO_WORD(CronEd.PR_TT*10));INTERN ASSIGN CronEd.PR.Setpoint[57]:=(REAL_TO_WORD(CronEd.PR_TT*10));INTERN ASSIGN CronEd.PR.Setpoint[56]:=(REAL_TO_WORD(CronEd.PR_TT*10))
rounded rectangle at (510,230)-(541,251): text "%.1f"; shows WORD_TO_REAL(CronEd.PR.Setpoint[60])/10; runs INTERN ASSIGN CronEd.PR.Setpoint[60]:=(REAL_TO_WORD(CronEd.PR_TT*10))
rounded rectangle at (510,250)-(541,271): text "%.1f"; shows WORD_TO_REAL(CronEd.PR.Setpoint[61])/10; runs INTERN ASSIGN CronEd.PR.Setpoint[61]:=(REAL_TO_WORD(CronEd.PR_TT*10))
rounded rectangle at (510,270)-(541,291): text "%.1f"; shows WORD_TO_REAL(CronEd.PR.Setpoint[62])/10; runs INTERN ASSIGN CronEd.PR.Setpoint[62]:=(REAL_TO_WORD(CronEd.PR_TT*10))
rounded rectangle at (510,290)-(541,311): text "%.1f"; shows WORD_TO_REAL(CronEd.PR.Setpoint[63])/10; runs INTERN ASSIGN CronEd.PR.Setpoint[63]:=(REAL_TO_WORD(CronEd.PR_TT*10))
rectangle at (510,200)-(541,221): text "h15"; runs INTERN ASSIGN CronEd.PR.Setpoint[63]:=(REAL_TO_WORD(CronEd.PR_TT*10));INTERN ASSIGN CronEd.PR.Setpoint[62]:=(REAL_TO_WORD(CronEd.PR_TT*10));INTERN ASSIGN CronEd.PR.Setpoint[61]:=(REAL_TO_WORD(CronEd.PR_TT*10));INTERN ASSIGN CronEd.PR.Setpoint[60]:=(REAL_TO_WORD(CronEd.PR_TT*10))
rounded rectangle at (540,230)-(571,251): text "%.1f"; shows WORD_TO_REAL(CronEd.PR.Setpoint[64])/10; runs INTERN ASSIGN CronEd.PR.Setpoint[64]:=(REAL_TO_WORD(CronEd.PR_TT*10))
rounded rectangle at (540,250)-(571,271): text "%.1f"; shows WORD_TO_REAL(CronEd.PR.Setpoint[65])/10; runs INTERN ASSIGN CronEd.PR.Setpoint[65]:=(REAL_TO_WORD(CronEd.PR_TT*10))
rounded rectangle at (540,270)-(571,291): text "%.1f"; shows WORD_TO_REAL(CronEd.PR.Setpoint[66])/10; runs INTERN ASSIGN CronEd.PR.Setpoint[66]:=(REAL_TO_WORD(CronEd.PR_TT*10))
rounded rectangle at (540,290)-(571,311): text "%.1f"; shows WORD_TO_REAL(CronEd.PR.Setpoint[67])/10; runs INTERN ASSIGN CronEd.PR.Setpoint[67]:=(REAL_TO_WORD(CronEd.PR_TT*10))
rectangle at (540,200)-(571,221): text "h16"; runs INTERN ASSIGN CronEd.PR.Setpoint[67]:=(REAL_TO_WORD(CronEd.PR_TT*10));INTERN ASSIGN CronEd.PR.Setpoint[66]:=(REAL_TO_WORD(CronEd.PR_TT*10));INTERN ASSIGN CronEd.PR.Setpoint[65]:=(REAL_TO_WORD(CronEd.PR_TT*10));INTERN ASSIGN CronEd.PR.Setpoint[64]:=(REAL_TO_WORD(CronEd.PR_TT*10))
rounded rectangle at (570,230)-(601,251): text "%.1f"; shows WORD_TO_REAL(CronEd.PR.Setpoint[68])/10; runs INTERN ASSIGN CronEd.PR.Setpoint[68]:=(REAL_TO_WORD(CronEd.PR_TT*10))
rounded rectangle at (570,250)-(601,271): text "%.1f"; shows WORD_TO_REAL(CronEd.PR.Setpoint[69])/10; runs INTERN ASSIGN CronEd.PR.Setpoint[69]:=(REAL_TO_WORD(CronEd.PR_TT*10))
rounded rectangle at (570,270)-(601,291): text "%.1f"; shows WORD_TO_REAL(CronEd.PR.Setpoint[70])/10; runs INTERN ASSIGN CronEd.PR.Setpoint[70]:=(REAL_TO_WORD(CronEd.PR_TT*10))
rounded rectangle at (570,290)-(601,311): text "%.1f"; shows WORD_TO_REAL(CronEd.PR.Setpoint[71])/10; runs INTERN ASSIGN CronEd.PR.Setpoint[71]:=(REAL_TO_WORD(CronEd.PR_TT*10))
rectangle at (570,200)-(601,221): text "h17"; runs INTERN ASSIGN CronEd.PR.Setpoint[71]:=(REAL_TO_WORD(CronEd.PR_TT*10));INTERN ASSIGN CronEd.PR.Setpoint[70]:=(REAL_TO_WORD(CronEd.PR_TT*10));INTERN ASSIGN CronEd.PR.Setpoint[69]:=(REAL_TO_WORD(CronEd.PR_TT*10));INTERN ASSIGN CronEd.PR.Setpoint[68]:=(REAL_TO_WORD(CronEd.PR_TT*10))
rounded rectangle at (600,230)-(631,251): text "%.1f"; shows WORD_TO_REAL(CronEd.PR.Setpoint[72])/10; runs INTERN ASSIGN CronEd.PR.Setpoint[72]:=(REAL_TO_WORD(CronEd.PR_TT*10))
rounded rectangle at (600,250)-(631,271): text "%.1f"; shows WORD_TO_REAL(CronEd.PR.Setpoint[73])/10; runs INTERN ASSIGN CronEd.PR.Setpoint[73]:=(REAL_TO_WORD(CronEd.PR_TT*10))
rounded rectangle at (600,270)-(631,291): text "%.1f"; shows WORD_TO_REAL(CronEd.PR.Setpoint[74])/10; runs INTERN ASSIGN CronEd.PR.Setpoint[74]:=(REAL_TO_WORD(CronEd.PR_TT*10))
rounded rectangle at (600,290)-(631,311): text "%.1f"; shows WORD_TO_REAL(CronEd.PR.Setpoint[75])/10; runs INTERN ASSIGN CronEd.PR.Setpoint[75]:=(REAL_TO_WORD(CronEd.PR_TT*10))
rectangle at (600,200)-(631,221): text "h18"; runs INTERN ASSIGN CronEd.PR.Setpoint[75]:=(REAL_TO_WORD(CronEd.PR_TT*10));INTERN ASSIGN CronEd.PR.Setpoint[74]:=(REAL_TO_WORD(CronEd.PR_TT*10));INTERN ASSIGN CronEd.PR.Setpoint[73]:=(REAL_TO_WORD(CronEd.PR_TT*10));INTERN ASSIGN CronEd.PR.Setpoint[72]:=(REAL_TO_WORD(CronEd.PR_TT*10))
rounded rectangle at (630,230)-(661,251): text "%.1f"; shows WORD_TO_REAL(CronEd.PR.Setpoint[76])/10; runs INTERN ASSIGN CronEd.PR.Setpoint[76]:=(REAL_TO_WORD(CronEd.PR_TT*10))
rounded rectangle at (630,250)-(661,271): text "%.1f"; shows WORD_TO_REAL(CronEd.PR.Setpoint[77])/10; runs INTERN ASSIGN CronEd.PR.Setpoint[77]:=(REAL_TO_WORD(CronEd.PR_TT*10))
rounded rectangle at (630,270)-(661,291): text "%.1f"; shows WORD_TO_REAL(CronEd.PR.Setpoint[78])/10; runs INTERN ASSIGN CronEd.PR.Setpoint[78]:=(REAL_TO_WORD(CronEd.PR_TT*10))
rounded rectangle at (630,290)-(661,311): text "%.1f"; shows WORD_TO_REAL(CronEd.PR.Setpoint[79])/10; runs INTERN ASSIGN CronEd.PR.Setpoint[79]:=(REAL_TO_WORD(CronEd.PR_TT*10))
rectangle at (630,200)-(661,221): text "h19"; runs INTERN ASSIGN CronEd.PR.Setpoint[79]:=(REAL_TO_WORD(CronEd.PR_TT*10));INTERN ASSIGN CronEd.PR.Setpoint[78]:=(REAL_TO_WORD(CronEd.PR_TT*10));INTERN ASSIGN CronEd.PR.Setpoint[77]:=(REAL_TO_WORD(CronEd.PR_TT*10));INTERN ASSIGN CronEd.PR.Setpoint[76]:=(REAL_TO_WORD(CronEd.PR_TT*10))
rounded rectangle at (660,230)-(691,251): text "%.1f"; shows WORD_TO_REAL(CronEd.PR.Setpoint[80])/10; runs INTERN ASSIGN CronEd.PR.Setpoint[80]:=(REAL_TO_WORD(CronEd.PR_TT*10))
rounded rectangle at (660,250)-(691,271): text "%.1f"; shows WORD_TO_REAL(CronEd.PR.Setpoint[81])/10; runs INTERN ASSIGN CronEd.PR.Setpoint[81]:=(REAL_TO_WORD(CronEd.PR_TT*10))
rounded rectangle at (660,270)-(691,291): text "%.1f"; shows WORD_TO_REAL(CronEd.PR.Setpoint[82])/10; runs INTERN ASSIGN CronEd.PR.Setpoint[82]:=(REAL_TO_WORD(CronEd.PR_TT*10))
rounded rectangle at (660,290)-(691,311): text "%.1f"; shows WORD_TO_REAL(CronEd.PR.Setpoint[83])/10; runs INTERN ASSIGN CronEd.PR.Setpoint[83]:=(REAL_TO_WORD(CronEd.PR_TT*10))
rectangle at (660,200)-(691,221): text "h20"; runs INTERN ASSIGN CronEd.PR.Setpoint[83]:=(REAL_TO_WORD(CronEd.PR_TT*10));INTERN ASSIGN CronEd.PR.Setpoint[82]:=(REAL_TO_WORD(CronEd.PR_TT*10));INTERN ASSIGN CronEd.PR.Setpoint[81]:=(REAL_TO_WORD(CronEd.PR_TT*10));INTERN ASSIGN CronEd.PR.Setpoint[80]:=(REAL_TO_WORD(CronEd.PR_TT*10))
rounded rectangle at (690,230)-(721,251): text "%.1f"; shows WORD_TO_REAL(CronEd.PR.Setpoint[84])/10; runs INTERN ASSIGN CronEd.PR.Setpoint[84]:=(REAL_TO_WORD(CronEd.PR_TT*10))
rounded rectangle at (690,250)-(721,271): text "%.1f"; shows WORD_TO_REAL(CronEd.PR.Setpoint[85])/10; runs INTERN ASSIGN CronEd.PR.Setpoint[85]:=(REAL_TO_WORD(CronEd.PR_TT*10))
rounded rectangle at (690,270)-(721,291): text "%.1f"; shows WORD_TO_REAL(CronEd.PR.Setpoint[86])/10; runs INTERN ASSIGN CronEd.PR.Setpoint[86]:=(REAL_TO_WORD(CronEd.PR_TT*10))
rounded rectangle at (690,290)-(721,311): text "%.1f"; shows WORD_TO_REAL(CronEd.PR.Setpoint[87])/10; runs INTERN ASSIGN CronEd.PR.Setpoint[87]:=(REAL_TO_WORD(CronEd.PR_TT*10))
rectangle at (690,200)-(721,221): text "h21"; runs INTERN ASSIGN CronEd.PR.Setpoint[87]:=(REAL_TO_WORD(CronEd.PR_TT*10));INTERN ASSIGN CronEd.PR.Setpoint[86]:=(REAL_TO_WORD(CronEd.PR_TT*10));INTERN ASSIGN CronEd.PR.Setpoint[85]:=(REAL_TO_WORD(CronEd.PR_TT*10));INTERN ASSIGN CronEd.PR.Setpoint[84]:=(REAL_TO_WORD(CronEd.PR_TT*10))
rounded rectangle at (720,230)-(751,251): text "%.1f"; shows WORD_TO_REAL(CronEd.PR.Setpoint[88])/10; runs INTERN ASSIGN CronEd.PR.Setpoint[88]:=(REAL_TO_WORD(CronEd.PR_TT*10))
rounded rectangle at (720,250)-(751,271): text "%.1f"; shows WORD_TO_REAL(CronEd.PR.Setpoint[89])/10; runs INTERN ASSIGN CronEd.PR.Setpoint[89]:=(REAL_TO_WORD(CronEd.PR_TT*10))
rounded rectangle at (720,270)-(751,291): text "%.1f"; shows WORD_TO_REAL(CronEd.PR.Setpoint[90])/10; runs INTERN ASSIGN CronEd.PR.Setpoint[90]:=(REAL_TO_WORD(CronEd.PR_TT*10))
rounded rectangle at (720,290)-(751,311): text "%.1f"; shows WORD_TO_REAL(CronEd.PR.Setpoint[91])/10; runs INTERN ASSIGN CronEd.PR.Setpoint[91]:=(REAL_TO_WORD(CronEd.PR_TT*10))
rectangle at (720,200)-(751,221): text "h22"; runs INTERN ASSIGN CronEd.PR.Setpoint[91]:=(REAL_TO_WORD(CronEd.PR_TT*10));INTERN ASSIGN CronEd.PR.Setpoint[90]:=(REAL_TO_WORD(CronEd.PR_TT*10));INTERN ASSIGN CronEd.PR.Setpoint[89]:=(REAL_TO_WORD(CronEd.PR_TT*10));INTERN ASSIGN CronEd.PR.Setpoint[88]:=(REAL_TO_WORD(CronEd.PR_TT*10))
rounded rectangle at (750,230)-(781,251): text "%.1f"; shows WORD_TO_REAL(CronEd.PR.Setpoint[92])/10; runs INTERN ASSIGN CronEd.PR.Setpoint[92]:=(REAL_TO_WORD(CronEd.PR_TT*10))
rounded rectangle at (750,250)-(781,271): text "%.1f"; shows WORD_TO_REAL(CronEd.PR.Setpoint[93])/10; runs INTERN ASSIGN CronEd.PR.Setpoint[93]:=(REAL_TO_WORD(CronEd.PR_TT*10))
rounded rectangle at (750,270)-(781,291): text "%.1f"; shows WORD_TO_REAL(CronEd.PR.Setpoint[94])/10; runs INTERN ASSIGN CronEd.PR.Setpoint[94]:=(REAL_TO_WORD(CronEd.PR_TT*10))
rounded rectangle at (750,290)-(781,311): text "%.1f"; shows WORD_TO_REAL(CronEd.PR.Setpoint[95])/10; runs INTERN ASSIGN CronEd.PR.Setpoint[95]:=(REAL_TO_WORD(CronEd.PR_TT*10))
rectangle at (750,200)-(781,221): text "h23"; runs INTERN ASSIGN CronEd.PR.Setpoint[95]:=(REAL_TO_WORD(CronEd.PR_TT*10));INTERN ASSIGN CronEd.PR.Setpoint[94]:=(REAL_TO_WORD(CronEd.PR_TT*10));INTERN ASSIGN CronEd.PR.Setpoint[93]:=(REAL_TO_WORD(CronEd.PR_TT*10));INTERN ASSIGN CronEd.PR.Setpoint[92]:=(REAL_TO_WORD(CronEd.PR_TT*10))
rectangle at (410,360)-(491,381): text "Month"
rectangle at (490,360)-(531,381): text "%d"; shows CronEd.CA_Sel; alarm colour if CronEd.CA_Sel<>CronEd.CA_Act; editable 1..12
rectangle at (410,390)-(491,411): text "Profile Nr."
rectangle at (490,390)-(531,411): text "%d"; shows CronEd.CA_TPR; editable 0..10
button at (540,360)-(601,381): text "Load"; toggles CronEd.CA_Load
button at (610,360)-(671,381): text "Save"; toggles CronEd.CA_Save
rounded rectangle at (160,360)-(191,381): text "%d"; shows CronEd.CA.Profile[0]; invisible if CronEd.CA_DayF>0; alarm colour if CronEd.CA.Profile[0]=0; runs INTERN ASSIGN CronEd.CA.Profile[0]:=(CronEd.CA_TPR)
rectangle at (120,360)-(151,381): text "1"
rounded rectangle at (190,360)-(221,381): text "%d"; shows CronEd.CA.Profile[1]; invisible if CronEd.CA_DayF>1; alarm colour if CronEd.CA.Profile[1]=0; runs INTERN ASSIGN CronEd.CA.Profile[1]:=(CronEd.CA_TPR)
rounded rectangle at (220,360)-(251,381): text "%d"; shows CronEd.CA.Profile[2]; invisible if CronEd.CA_DayF>2; alarm colour if CronEd.CA.Profile[2]=0; runs INTERN ASSIGN CronEd.CA.Profile[2]:=(CronEd.CA_TPR)
rounded rectangle at (250,360)-(281,381): text "%d"; shows CronEd.CA.Profile[3]; invisible if CronEd.CA_DayF>3; alarm colour if CronEd.CA.Profile[3]=0; runs INTERN ASSIGN CronEd.CA.Profile[3]:=(CronEd.CA_TPR)
rounded rectangle at (280,360)-(311,381): text "%d"; shows CronEd.CA.Profile[4]; invisible if CronEd.CA_DayF>4; alarm colour if CronEd.CA.Profile[4]=0; runs INTERN ASSIGN CronEd.CA.Profile[4]:=(CronEd.CA_TPR)
rounded rectangle at (310,360)-(341,381): text "%d"; shows CronEd.CA.Profile[5]; invisible if CronEd.CA_DayF>5; alarm colour if CronEd.CA.Profile[5]=0; runs INTERN ASSIGN CronEd.CA.Profile[5]:=(CronEd.CA_TPR)
rounded rectangle at (340,360)-(371,381): text "%d"; shows CronEd.CA.Profile[6]; alarm colour if CronEd.CA.Profile[6]=0; runs INTERN ASSIGN CronEd.CA.Profile[6]:=(CronEd.CA_TPR)
rounded rectangle at (160,380)-(191,401): text "%d"; shows CronEd.CA.Profile[7]; alarm colour if CronEd.CA.Profile[7]=0; runs INTERN ASSIGN CronEd.CA.Profile[7]:=(CronEd.CA_TPR)
rectangle at (120,380)-(151,401): text "8"
rounded rectangle at (190,380)-(221,401): text "%d"; shows CronEd.CA.Profile[8]; alarm colour if CronEd.CA.Profile[8]=0; runs INTERN ASSIGN CronEd.CA.Profile[8]:=(CronEd.CA_TPR)
rounded rectangle at (220,380)-(251,401): text "%d"; shows CronEd.CA.Profile[9]; alarm colour if CronEd.CA.Profile[9]=0; runs INTERN ASSIGN CronEd.CA.Profile[9]:=(CronEd.CA_TPR)
rounded rectangle at (250,380)-(281,401): text "%d"; shows CronEd.CA.Profile[10]; alarm colour if CronEd.CA.Profile[10]=0; runs INTERN ASSIGN CronEd.CA.Profile[10]:=(CronEd.CA_TPR)
rounded rectangle at (280,380)-(311,401): text "%d"; shows CronEd.CA.Profile[11]; alarm colour if CronEd.CA.Profile[11]=0; runs INTERN ASSIGN CronEd.CA.Profile[11]:=(CronEd.CA_TPR)
rounded rectangle at (310,380)-(341,401): text "%d"; shows CronEd.CA.Profile[12]; alarm colour if CronEd.CA.Profile[12]=0; runs INTERN ASSIGN CronEd.CA.Profile[12]:=(CronEd.CA_TPR)
rounded rectangle at (340,380)-(371,401): text "%d"; shows CronEd.CA.Profile[13]; alarm colour if CronEd.CA.Profile[13]=0; runs INTERN ASSIGN CronEd.CA.Profile[13]:=(CronEd.CA_TPR)
rounded rectangle at (160,400)-(191,421): text "%d"; shows CronEd.CA.Profile[14]; alarm colour if CronEd.CA.Profile[14]=0; runs INTERN ASSIGN CronEd.CA.Profile[14]:=(CronEd.CA_TPR)
rectangle at (120,400)-(151,421): text "15"
rounded rectangle at (190,400)-(221,421): text "%d"; shows CronEd.CA.Profile[15]; alarm colour if CronEd.CA.Profile[15]=0; runs INTERN ASSIGN CronEd.CA.Profile[15]:=(CronEd.CA_TPR)
rounded rectangle at (220,400)-(251,421): text "%d"; shows CronEd.CA.Profile[16]; alarm colour if CronEd.CA.Profile[16]=0; runs INTERN ASSIGN CronEd.CA.Profile[16]:=(CronEd.CA_TPR)
rounded rectangle at (250,400)-(281,421): text "%d"; shows CronEd.CA.Profile[17]; alarm colour if CronEd.CA.Profile[17]=0; runs INTERN ASSIGN CronEd.CA.Profile[17]:=(CronEd.CA_TPR)
rounded rectangle at (280,400)-(311,421): text "%d"; shows CronEd.CA.Profile[18]; alarm colour if CronEd.CA.Profile[18]=0; runs INTERN ASSIGN CronEd.CA.Profile[18]:=(CronEd.CA_TPR)
rounded rectangle at (310,400)-(341,421): text "%d"; shows CronEd.CA.Profile[19]; alarm colour if CronEd.CA.Profile[19]=0; runs INTERN ASSIGN CronEd.CA.Profile[19]:=(CronEd.CA_TPR)
rounded rectangle at (340,400)-(371,421): text "%d"; shows CronEd.CA.Profile[20]; alarm colour if CronEd.CA.Profile[20]=0; runs INTERN ASSIGN CronEd.CA.Profile[20]:=(CronEd.CA_TPR)
rounded rectangle at (160,420)-(191,441): text "%d"; shows CronEd.CA.Profile[21]; alarm colour if CronEd.CA.Profile[21]=0; runs INTERN ASSIGN CronEd.CA.Profile[21]:=(CronEd.CA_TPR)
rectangle at (120,420)-(151,441): text "22"
rounded rectangle at (190,420)-(221,441): text "%d"; shows CronEd.CA.Profile[22]; alarm colour if CronEd.CA.Profile[22]=0; runs INTERN ASSIGN CronEd.CA.Profile[22]:=(CronEd.CA_TPR)
rounded rectangle at (220,420)-(251,441): text "%d"; shows CronEd.CA.Profile[23]; alarm colour if CronEd.CA.Profile[23]=0; runs INTERN ASSIGN CronEd.CA.Profile[23]:=(CronEd.CA_TPR)
rounded rectangle at (250,420)-(281,441): text "%d"; shows CronEd.CA.Profile[24]; alarm colour if CronEd.CA.Profile[24]=0; runs INTERN ASSIGN CronEd.CA.Profile[24]:=(CronEd.CA_TPR)
rounded rectangle at (280,420)-(311,441): text "%d"; shows CronEd.CA.Profile[25]; alarm colour if CronEd.CA.Profile[25]=0; runs INTERN ASSIGN CronEd.CA.Profile[25]:=(CronEd.CA_TPR)
rounded rectangle at (310,420)-(341,441): text "%d"; shows CronEd.CA.Profile[26]; alarm colour if CronEd.CA.Profile[26]=0; runs INTERN ASSIGN CronEd.CA.Profile[26]:=(CronEd.CA_TPR)
rounded rectangle at (340,420)-(371,441): text "%d"; shows CronEd.CA.Profile[27]; alarm colour if CronEd.CA.Profile[27]=0; runs INTERN ASSIGN CronEd.CA.Profile[27]:=(CronEd.CA_TPR)
rounded rectangle at (160,440)-(191,461): text "%d"; shows CronEd.CA.Profile[28]; alarm colour if CronEd.CA.Profile[28]=0; runs INTERN ASSIGN CronEd.CA.Profile[28]:=(CronEd.CA_TPR)
rectangle at (120,440)-(151,461): text "29"
rounded rectangle at (190,440)-(221,461): text "%d"; shows CronEd.CA.Profile[29]; alarm colour if CronEd.CA.Profile[29]=0; runs INTERN ASSIGN CronEd.CA.Profile[29]:=(CronEd.CA_TPR)
rounded rectangle at (220,440)-(251,461): text "%d"; shows CronEd.CA.Profile[30]; alarm colour if CronEd.CA.Profile[30]=0; runs INTERN ASSIGN CronEd.CA.Profile[30]:=(CronEd.CA_TPR)
rounded rectangle at (250,440)-(281,461): text "%d"; shows CronEd.CA.Profile[31]; alarm colour if CronEd.CA.Profile[31]=0; runs INTERN ASSIGN CronEd.CA.Profile[31]:=(CronEd.CA_TPR)
rounded rectangle at (280,440)-(311,461): text "%d"; shows CronEd.CA.Profile[32]; invisible if CronEd.CA_DayL<32; alarm colour if CronEd.CA.Profile[32]=0; runs INTERN ASSIGN CronEd.CA.Profile[32]:=(CronEd.CA_TPR)
rounded rectangle at (310,440)-(341,461): text "%d"; shows CronEd.CA.Profile[33]; invisible if CronEd.CA_DayL<33; alarm colour if CronEd.CA.Profile[33]=0; runs INTERN ASSIGN CronEd.CA.Profile[33]:=(CronEd.CA_TPR)
rounded rectangle at (340,440)-(371,461): text "%d"; shows CronEd.CA.Profile[34]; invisible if CronEd.CA_DayL<34; alarm colour if CronEd.CA.Profile[34]=0; runs INTERN ASSIGN CronEd.CA.Profile[34]:=(CronEd.CA_TPR)
rounded rectangle at (160,460)-(191,481): text "%d"; shows CronEd.CA.Profile[35]; invisible if CronEd.CA_DayL<35; alarm colour if CronEd.CA.Profile[35]=0; runs INTERN ASSIGN CronEd.CA.Profile[35]:=(CronEd.CA_TPR)
rectangle at (120,460)-(151,481): text "36"; invisible if CronEd.CA_DayL<35
rounded rectangle at (190,460)-(221,481): text "%d"; shows CronEd.CA.Profile[36]; invisible if CronEd.CA_DayL<36; alarm colour if CronEd.CA.Profile[36]=0; runs INTERN ASSIGN CronEd.CA.Profile[36]:=(CronEd.CA_TPR)
rounded rectangle at (220,460)-(251,481): text "%d"; shows CronEd.CA.Profile[37]; invisible if CronEd.CA_DayL<37; alarm colour if CronEd.CA.Profile[37]=0; runs INTERN ASSIGN CronEd.CA.Profile[37]:=(CronEd.CA_TPR)
rounded rectangle at (250,460)-(281,481): text "%d"; shows CronEd.CA.Profile[38]; invisible if CronEd.CA_DayL<38; alarm colour if CronEd.CA.Profile[38]=0; runs INTERN ASSIGN CronEd.CA.Profile[38]:=(CronEd.CA_TPR)
rounded rectangle at (280,460)-(311,481): text "%d"; shows CronEd.CA.Profile[39]; invisible if CronEd.CA_DayL<39; alarm colour if CronEd.CA.Profile[39]=0; runs INTERN ASSIGN CronEd.CA.Profile[39]:=(CronEd.CA_TPR)
rounded rectangle at (310,460)-(341,481): text "%d"; shows CronEd.CA.Profile[40]; invisible if CronEd.CA_DayL<40; alarm colour if CronEd.CA.Profile[40]=0; runs INTERN ASSIGN CronEd.CA.Profile[40]:=(CronEd.CA_TPR)
rounded rectangle at (340,460)-(371,481): text "%d"; shows CronEd.CA.Profile[41]; invisible if CronEd.CA_DayL<41; alarm colour if CronEd.CA.Profile[41]=0; runs INTERN ASSIGN CronEd.CA.Profile[41]:=(CronEd.CA_TPR)
rectangle at (310,60)-(371,81): text "Year"
rectangle at (370,60)-(411,81): text "%d"; shows CronEd.CN_YSel; alarm colour if CronEd.CN_YSel<>CronEd.CN_YAct; editable 2000..2100
rectangle at (480,60)-(761,81): text "%s"; shows CronEd.Message
button at (10,50)-(71,81): text "REINIT"; runs INTERN ASSIGN CRON03.InitOK:=(FALSE);INTERN ASSIGN CRON04.InitOK:=(FALSE);INTERN ASSIGN CRON05.InitOK:=(FALSE);INTERN ASSIGN CRON06.InitOK:=(FALSE);INTERN ASSIGN CRON01.InitOK:=(FALSE)
2 more shapes without text or variables
*)
